KUKA KRL program: MyProgram_196().src

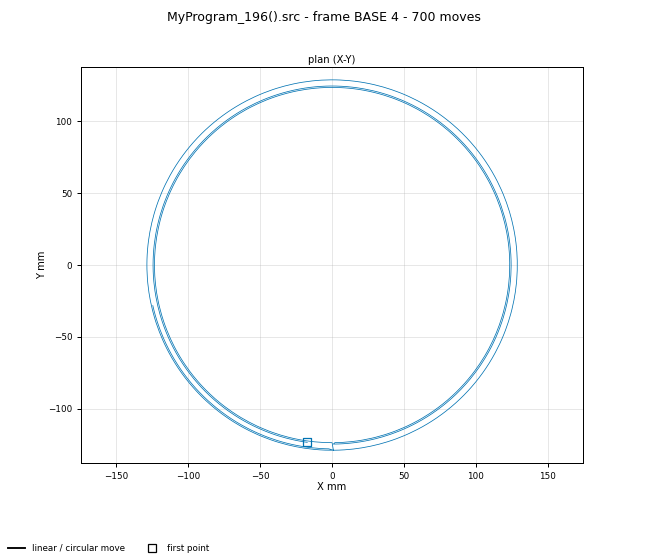
[picture p0: tool path of MyProgram_196().src in frame BASE 4, 700 of 700 moves have a stored position in this frame; points joined in program order, loops and branches not executed]
&ACCESS RVP
&REL 1
&PARAM TEMPLATE = C:\KRC\Roboter\Template\vorgabe
&PARAM EDITMASK = *
DEF MyProgram_196()
; ---- Setting reference (Base) ----
$BASE = BASE_DATA[4]

; --------------------------
; ---- Setting tool (TCP) ----
$TOOL = TOOL_DATA[3]
; --------------------------

$VEL.CP = VEL_APROX_PRINT
Startdeposition()
$VEL.CP = VEL_PRINT
LIN {X -17.3066,Y -123.2916,Z 141,A -101.2805,B 23.689,C -1.1574,E1 23.6926,E2 548.0217} C_DIS
LIN {X -20.7181,Y -122.7642,Z 141,A -102.9129,B 23.689,C -1.1559,E1 23.6881,E2 549.6594} C_DIS
LIN {X -25.1482,Y -121.934,Z 141,A -104.9652,B 23.689,C -1.1577,E1 23.6825,E2 551.7095} C_DIS
LIN {X -31.1595,Y -120.5388,Z 141,A -107.6921,B 23.6887,C -1.1643,E1 23.6751,E2 554.424} C_DIS
LIN {X -33.6692,Y -119.8608,Z 141,A -108.9963,B 23.6889,C -1.1602,E1 23.6716,E2 555.7403} C_DIS
LIN {X -36.6545,Y -118.9819,Z 141,A -110.4119,B 23.6889,C -1.162,E1 23.6678,E2 557.1541} C_DIS
LIN {X -39.4614,Y -118.0805,Z 141,A -111.8065,B 23.6889,C -1.1614,E1 23.6641,E2 558.5529} C_DIS
LIN {X -42.5428,Y -117.006,Z 141,A -113.362,B 23.6889,C -1.1604,E1 23.66,E2 560.1144} C_DIS
LIN {X -46.169,Y -115.6234,Z 141,A -115.2404,B 23.6889,C -1.158,E1 23.6551,E2 562.0028} C_DIS
LIN {X -50.7496,Y -113.6867,Z 141,A -117.3609,B 23.6885,C -1.1679,E1 23.6497,E2 564.1039} C_DIS
LIN {X -54.336,Y -112.0192,Z 141,A -119.1495,B 23.6884,C -1.1715,E1 23.6452,E2 565.8885} C_DIS
LIN {X -57.8725,Y -110.2313,Z 141,A -120.9361,B 23.6882,C -1.1755,E1 23.6407,E2 567.6703} C_DIS
LIN {X -61.1046,Y -108.4752,Z 141,A -122.7725,B 23.6884,C -1.1715,E1 23.6362,E2 569.5223} C_DIS
LIN {X -64.9923,Y -106.1916,Z 141,A -124.5928,B 23.6877,C -1.1857,E1 23.6319,E2 571.313} C_DIS
LIN {X -67.5246,Y -104.6,Z 141,A -126.2397,B 23.6882,C -1.176,E1 23.628,E2 572.9897} C_DIS
LIN {X -71.7527,Y -101.7456,Z 141,A -128.2349,B 23.6872,C -1.1952,E1 23.6235,E2 574.9438} C_DIS
LIN {X -75.0263,Y -99.3563,Z 141,A -130.4687,B 23.6879,C -1.1824,E1 23.6183,E2 577.218} C_DIS
LIN {X -78.4831,Y -96.6498,Z 141,A -132.5143,B 23.6877,C -1.1851,E1 23.6139,E2 579.2651} C_DIS
LIN {X -81.6923,Y -93.9523,Z 141,A -134.4843,B 23.6877,C -1.1871,E1 23.6097,E2 581.2382} C_DIS
LIN {X -85.1342,Y -90.8457,Z 141,A -136.6203,B 23.6874,C -1.1913,E1 23.6053,E2 583.3728} C_DIS
LIN {X -88.2078,Y -87.8637,Z 141,A -138.5647,B 23.6872,C -1.1967,E1 23.6014,E2 585.3126} C_DIS
LIN {X -91.1663,Y -84.79,Z 141,A -140.5025,B 23.6869,C -1.2021,E1 23.5977,E2 587.2457} C_DIS
LIN {X -94.3561,Y -81.2253,Z 141,A -142.5001,B 23.6863,C -1.2158,E1 23.5941,E2 589.2185} C_DIS
LIN {X -96.0854,Y -79.1726,Z 141,A -144.0072,B 23.6867,C -1.2071,E1 23.5913,E2 590.7547} C_DIS
LIN {X -98.6893,Y -75.9024,Z 141,A -145.9776,B 23.6866,C -1.2098,E1 23.5879,E2 592.7283} C_DIS
LIN {X -101.3019,Y -72.3779,Z 141,A -148.129,B 23.6866,C -1.2092,E1 23.5844,E2 594.8922} C_DIS
LIN {X -103.9608,Y -68.5039,Z 141,A -150.1422,B 23.686,C -1.2211,E1 23.5813,E2 596.8864} C_DIS
LIN {X -106.2239,Y -64.9397,Z 141,A -152.0556,B 23.6857,C -1.2275,E1 23.5785,E2 598.7942} C_DIS
LIN {X -108.3531,Y -61.3219,Z 141,A -154.0839,B 23.6857,C -1.2286,E1 23.5756,E2 600.8308} C_DIS
LIN {X -110.493,Y -57.374,Z 141,A -155.9511,B 23.6849,C -1.2428,E1 23.5732,E2 602.6732} C_DIS
LIN {X -112.6362,Y -53.0445,Z 141,A -158.2325,B 23.6848,C -1.2465,E1 23.5704,E2 604.9581} C_DIS
LIN {X -114.2456,Y -49.4785,Z 141,A -160.0905,B 23.6846,C -1.2493,E1 23.5683,E2 606.82} C_DIS
LIN {X -115.6132,Y -46.1941,Z 141,A -161.8382,B 23.6846,C -1.2495,E1 23.5664,E2 608.5777} C_DIS
LIN {X -117.0709,Y -42.3627,Z 141,A -163.641,B 23.6842,C -1.2586,E1 23.5647,E2 610.3685} C_DIS
LIN {X -118.1962,Y -39.114,Z 141,A -165.24,B 23.684,C -1.2626,E1 23.5632,E2 611.967} C_DIS
LIN {X -119.7022,Y -34.2364,Z 141,A -167.5392,B 23.6835,C -1.2718,E1 23.5614,E2 614.2573} C_DIS
LIN {X -120.5071,Y -31.2844,Z 141,A -168.9347,B 23.6832,C -1.2767,E1 23.5604,E2 615.6491} C_DIS
LIN {X -121.2131,Y -28.4269,Z 141,A -170.8638,B 23.6842,C -1.257,E1 23.5591,E2 617.6396} C_DIS
LIN {X -122.0549,Y -24.5539,Z 141,A -171.9959,B 23.6825,C -1.2915,E1 23.5585,E2 618.6924} C_DIS
LIN {X -122.5458,Y -21.9722,Z 141,A -173.9291,B 23.6838,C -1.2653,E1 23.5575,E2 620.7035} C_DIS
LIN {X -123.2084,Y -17.8892,Z 141,A -175.3683,B 23.6825,C -1.2905,E1 23.557,E2 622.0886} C_DIS
LIN {X -123.6579,Y -14.4595,Z 141,A -176.892,B 23.6821,C -1.2984,E1 23.5564,E2 623.6022} C_DIS
LIN {X -123.9664,Y -11.5209,Z 141,A -178.4267,B 23.6823,C -1.2955,E1 23.556,E2 625.1539} C_DIS
LIN {X -124.2836,Y -7.3465,Z 141,A 179.8305,B 23.6816,C -1.3093,E1 23.5557,E2 626.8732} C_DIS
LIN {X -124.4226,Y -4.4158,Z 141,A 178.2604,B 23.6818,C -1.3046,E1 23.5555,E2 628.4653} C_DIS
LIN {X -124.5041,Y 0,Z 141,A 176.192,B 23.6815,C -1.3096,E1 23.5555,E2 630.5343} C_DIS
LIN {X -124.4406,Y 3.8734,Z 141,A 174.6213,B 23.6808,C -1.3242,E1 23.5555,E2 632.0784} C_DIS
LIN {X -124.2882,Y 7.271,Z 141,A 172.9166,B 23.6808,C -1.3235,E1 23.5558,E2 633.7958} C_DIS
LIN {X -124.0047,Y 11.1136,Z 141,A 170.7128,B 23.6815,C -1.3115,E1 23.5563,E2 636.0437} C_DIS
LIN {X -123.6032,Y 14.9174,Z 141,A 168.4748,B 23.6822,C -1.2977,E1 23.5571,E2 638.3305} C_DIS
LIN {X -122.7092,Y 21.0481,Z 141,A 166.196,B 23.6805,C -1.3303,E1 23.5581,E2 640.542} C_DIS
LIN {X -122.1083,Y 24.2919,Z 141,A 164.8985,B 23.6797,C -1.3443,E1 23.5588,E2 641.8126} C_DIS
LIN {X -121.1947,Y 28.503,Z 141,A 162.8874,B 23.6794,C -1.3495,E1 23.56,E2 643.8233} C_DIS
LIN {X -120.2681,Y 32.1841,Z 141,A 161.2198,B 23.679,C -1.3583,E1 23.5612,E2 645.4791} C_DIS
LIN {X -119.4143,Y 35.2207,Z 141,A 159.7511,B 23.6788,C -1.3622,E1 23.5623,E2 646.947} C_DIS
LIN {X -118.4127,Y 38.4576,Z 141,A 158.2228,B 23.6784,C -1.3684,E1 23.5636,E2 648.4692} C_DIS
LIN {X -117.5027,Y 41.1515,Z 141,A 156.9647,B 23.6781,C -1.3746,E1 23.5648,E2 649.7193} C_DIS
LIN {X -116.5143,Y 43.8707,Z 141,A 155.022,B 23.6792,C -1.3535,E1 23.5667,E2 651.7266} C_DIS
LIN {X -114.9502,Y 47.8189,Z 141,A 153.8518,B 23.6771,C -1.3919,E1 23.5679,E2 652.8074} C_DIS
LIN {X -113.6029,Y 50.9369,Z 141,A 151.9527,B 23.6776,C -1.3827,E1 23.57,E2 654.7407} C_DIS
LIN {X -112.2654,Y 53.8206,Z 141,A 150.502,B 23.6774,C -1.3876,E1 23.5718,E2 656.1875} C_DIS
LIN {X -110.5566,Y 57.2529,Z 141,A 148.7321,B 23.6771,C -1.3926,E1 23.574,E2 657.955} C_DIS
LIN {X -108.919,Y 60.3099,Z 141,A 146.6227,B 23.678,C -1.376,E1 23.5769,E2 660.1177} C_DIS
LIN {X -106.7792,Y 64.0229,Z 141,A 145.3003,B 23.6762,C -1.4086,E1 23.5787,E2 661.3657} C_DIS
LIN {X -105.139,Y 66.682,Z 141,A 143.6415,B 23.6765,C -1.4035,E1 23.5812,E2 663.0464} C_DIS
LIN {X -102.8195,Y 70.2058,Z 141,A 141.6627,B 23.6763,C -1.4074,E1 23.5842,E2 665.0259} C_DIS
LIN {X -100.2413,Y 73.8399,Z 141,A 139.749,B 23.6756,C -1.4187,E1 23.5873,E2 666.9211} C_DIS
LIN {X -98.1212,Y 76.6353,Z 141,A 137.9549,B 23.6758,C -1.4155,E1 23.5904,E2 668.7323} C_DIS
LIN {X -95.2628,Y 80.1602,Z 141,A 135.9027,B 23.6754,C -1.4225,E1 23.5941,E2 670.777} C_DIS
LIN {X -92.4463,Y 83.3933,Z 141,A 133.9366,B 23.6751,C -1.4278,E1 23.5977,E2 672.7392} C_DIS
LIN {X -89.5628,Y 86.4821,Z 141,A 131.9927,B 23.6748,C -1.4327,E1 23.6014,E2 674.6799} C_DIS
LIN {X -86.8396,Y 89.2167,Z 141,A 130.1509,B 23.6748,C -1.4342,E1 23.6051,E2 676.5262} C_DIS
LIN {X -83.8458,Y 92.0357,Z 141,A 128.2976,B 23.6744,C -1.4403,E1 23.6089,E2 678.3723} C_DIS
LIN {X -80.2512,Y 95.1865,Z 141,A 126.0391,B 23.6743,C -1.4428,E1 23.6136,E2 680.6339} C_DIS
LIN {X -76.8712,Y 97.936,Z 141,A 124.0446,B 23.674,C -1.4476,E1 23.618,E2 682.6243} C_DIS
LIN {X -73.4057,Y 100.5603,Z 141,A 121.9863,B 23.6739,C -1.4493,E1 23.6226,E2 684.6862} C_DIS
LIN {X -69.956,Y 102.9894,Z 141,A 120.0614,B 23.6736,C -1.4539,E1 23.627,E2 686.6065} C_DIS
LIN {X -66.1231,Y 105.4917,Z 141,A 117.6109,B 23.6742,C -1.4433,E1 23.6329,E2 689.0918} C_DIS
LIN {X -62.8782,Y 107.457,Z 141,A 115.78,B 23.6742,C -1.4428,E1 23.6373,E2 690.9298} C_DIS
LIN {X -59.2115,Y 109.5205,Z 141,A 114.2417,B 23.6731,C -1.463,E1 23.641,E2 692.4221} C_DIS
LIN {X -53.1473,Y 112.5871,Z 141,A 111.2946,B 23.6723,C -1.4758,E1 23.6483,E2 695.3456} C_DIS
LIN {X -50.7226,Y 113.6987,Z 141,A 109.9492,B 23.6725,C -1.4726,E1 23.6517,E2 696.7024} C_DIS
LIN {X -47.7132,Y 114.9944,Z 141,A 108.542,B 23.6721,C -1.4791,E1 23.6553,E2 698.0969} C_DIS
LIN {X -45.0235,Y 116.0736,Z 141,A 107.0366,B 23.6725,C -1.4735,E1 23.6593,E2 699.6198} C_DIS
LIN {X -41.6006,Y 117.3457,Z 141,A 105.0029,B 23.6732,C -1.4603,E1 23.6647,E2 701.6905} C_DIS
LIN {X -38.0606,Y 118.5395,Z 141,A 103.7953,B 23.6718,C -1.4845,E1 23.6678,E2 702.8401} C_DIS
LIN {X -34.6323,Y 119.5865,Z 141,A 102.079,B 23.6718,C -1.4834,E1 23.6724,E2 704.5622} C_DIS
LIN {X -30.8263,Y 120.6234,Z 141,A 99.7305,B 23.6731,C -1.4621,E1 23.6789,E2 706.9675} C_DIS
LIN {X -26.6986,Y 121.6043,Z 141,A 98.4667,B 23.6713,C -1.4938,E1 23.6821,E2 708.154} C_DIS
LIN {X -22.8887,Y 122.3789,Z 141,A 96.3822,B 23.672,C -1.4823,E1 23.6879,E2 710.2696} C_DIS
LIN {X -18.9799,Y 123.0448,Z 141,A 94.6737,B 23.6716,C -1.4887,E1 23.6926,E2 711.9638} C_DIS
LIN {X -15.2406,Y 123.5647,Z 141,A 92.9076,B 23.6716,C -1.4885,E1 23.6975,E2 713.7319} C_DIS
LIN {X -11.7063,Y 123.9486,Z 141,A 91.3468,B 23.6713,C -1.4927,E1 23.7018,E2 715.2833} C_DIS
LIN {X -8.1197,Y 124.2359,Z 141,A 89.5749,B 23.6716,C -1.4882,E1 23.7067,E2 717.067} C_DIS
LIN {X -4.0364,Y 124.4361,Z 141,A 87.8019,B 23.6713,C -1.4936,E1 23.7117,E2 718.827} C_DIS
LIN {X -1.1493,Y 124.4958,Z 141,A 86.3456,B 23.6716,C -1.4883,E1 23.7158,E2 720.2966} C_DIS
LIN {X 2.7069,Y 124.4724,Z 141,A 84.5293,B 23.6716,C -1.4866,E1 23.7208,E2 722.1168} C_DIS
LIN {X 6.669,Y 124.3221,Z 141,A 82.715,B 23.6716,C -1.4872,E1 23.7259,E2 723.929} C_DIS
LIN {X 10.5326,Y 124.0538,Z 141,A 81.0523,B 23.6714,C -1.4924,E1 23.7305,E2 725.5778} C_DIS
LIN {X 14.2232,Y 123.686,Z 141,A 79.2934,B 23.6715,C -1.4898,E1 23.7354,E2 727.342} C_DIS
LIN {X 17.7081,Y 123.2343,Z 141,A 77.6949,B 23.6715,C -1.4902,E1 23.7398,E2 728.9379} C_DIS
LIN {X 22.0126,Y 122.5385,Z 141,A 75.6852,B 23.6715,C -1.4894,E1 23.7453,E2 730.9475} C_DIS
LIN {X 28.4618,Y 121.2037,Z 141,A 72.786,B 23.6713,C -1.4938,E1 23.7532,E2 733.8318} C_DIS
LIN {X 31.9757,Y 120.3236,Z 141,A 71.0084,B 23.6716,C -1.4878,E1 23.7581,E2 735.6216} C_DIS
LIN {X 35.5975,Y 119.3039,Z 141,A 69.3551,B 23.6715,C -1.49,E1 23.7625,E2 737.2662} C_DIS
LIN {X 38.629,Y 118.3577,Z 141,A 67.8802,B 23.6716,C -1.4882,E1 23.7664,E2 738.7427} C_DIS
LIN {X 41.7416,Y 117.2949,Z 141,A 66.3878,B 23.6716,C -1.4879,E1 23.7703,E2 740.2328} C_DIS
LIN {X 45.712,Y 115.8059,Z 141,A 64.4266,B 23.6718,C -1.4855,E1 23.7754,E2 742.1954} C_DIS
LIN {X 48.1386,Y 114.8167,Z 141,A 63.1889,B 23.6719,C -1.4828,E1 23.7786,E2 743.4368} C_DIS
LIN {X 51.6422,Y 113.2859,Z 141,A 61.4616,B 23.6719,C -1.4822,E1 23.783,E2 745.1611} C_DIS
LIN {X 55.6591,Y 111.3671,Z 141,A 59.4544,B 23.6719,C -1.4816,E1 23.7881,E2 747.1642} C_DIS
LIN {X 59.597,Y 109.3107,Z 141,A 57.1094,B 23.673,C -1.4649,E1 23.7939,E2 749.5435} C_DIS
LIN {X 63.4067,Y 107.1465,Z 141,A 55.2096,B 23.6728,C -1.4673,E1 23.7985,E2 751.4312} C_DIS
LIN {X 66.7928,Y 105.0691,Z 141,A 53.3736,B 23.673,C -1.4641,E1 23.8029,E2 753.269} C_DIS
LIN {X 70.403,Y 102.6842,Z 141,A 51.4427,B 23.673,C -1.4636,E1 23.8073,E2 755.1942} C_DIS
LIN {X 73.2476,Y 100.6751,Z 141,A 49.9898,B 23.6728,C -1.4678,E1 23.8106,E2 756.6313} C_DIS
LIN {X 75.9908,Y 98.6212,Z 141,A 48.3246,B 23.6732,C -1.4609,E1 23.8143,E2 758.3073} C_DIS
LIN {X 79.7633,Y 95.5958,Z 141,A 46.0146,B 23.6737,C -1.4527,E1 23.8193,E2 760.6284} C_DIS
LIN {X 83.2093,Y 92.6115,Z 141,A 43.9696,B 23.6737,C -1.451,E1 23.8236,E2 762.669} C_DIS
LIN {X 86.3521,Y 89.6887,Z 141,A 41.9825,B 23.6741,C -1.4463,E1 23.8276,E2 764.6591} C_DIS
LIN {X 89.3005,Y 86.753,Z 141,A 40.1226,B 23.6741,C -1.4447,E1 23.8313,E2 766.5145} C_DIS
LIN {X 91.9746,Y 83.9131,Z 141,A 38.2695,B 23.6745,C -1.4379,E1 23.8348,E2 768.3758} C_DIS
LIN {X 94.9716,Y 80.505,Z 141,A 36.2299,B 23.6747,C -1.4354,E1 23.8385,E2 770.4119} C_DIS
LIN {X 97.6729,Y 77.2061,Z 141,A 34.236,B 23.675,C -1.4291,E1 23.842,E2 772.4113} C_DIS
LIN {X 100.3932,Y 73.6331,Z 141,A 32.3813,B 23.6747,C -1.4341,E1 23.8451,E2 774.2443} C_DIS
LIN {X 102.6283,Y 70.4845,Z 141,A 30.4624,B 23.6754,C -1.4228,E1 23.8482,E2 776.1812} C_DIS
LIN {X 104.9443,Y 66.9877,Z 141,A 28.5479,B 23.6756,C -1.4185,E1 23.8511,E2 778.0963} C_DIS
LIN {X 107.5449,Y 62.7282,Z 141,A 26.2165,B 23.6761,C -1.4107,E1 23.8545,E2 780.4343} C_DIS
LIN {X 109.7049,Y 58.8682,Z 141,A 24.1542,B 23.6765,C -1.4038,E1 23.8573,E2 782.5022} C_DIS
LIN {X 111.8497,Y 54.6808,Z 141,A 22.2107,B 23.6762,C -1.4084,E1 23.8597,E2 784.4234} C_DIS
LIN {X 113.1798,Y 51.8717,Z 141,A 20.8015,B 23.6764,C -1.4053,E1 23.8613,E2 785.8321} C_DIS
LIN {X 114.4208,Y 49.0733,Z 141,A 19.3376,B 23.6768,C -1.3986,E1 23.863,E2 787.3042} C_DIS
LIN {X 116.0662,Y 45.0425,Z 141,A 17.3425,B 23.6771,C -1.3931,E1 23.865,E2 789.3011} C_DIS
LIN {X 117.4217,Y 41.3853,Z 141,A 15.3627,B 23.6778,C -1.3788,E1 23.8669,E2 791.3045} C_DIS
LIN {X 119.9692,Y 33.2816,Z 141,A 11.7012,B 23.6778,C -1.3788,E1 23.8699,E2 794.9438} C_DIS
LIN {X 120.5954,Y 30.9366,Z 141,A 10.3603,B 23.6786,C -1.3646,E1 23.8709,E2 796.3118} C_DIS
LIN {X 121.5379,Y 27.0058,Z 141,A 8.775,B 23.6782,C -1.3721,E1 23.8718,E2 797.8689} C_DIS
LIN {X 122.4429,Y 22.5467,Z 141,A 6.549,B 23.6789,C -1.3591,E1 23.873,E2 800.1132} C_DIS
LIN {X 123.0538,Y 18.9216,Z 141,A 4.9728,B 23.6789,C -1.3593,E1 23.8737,E2 801.6789} C_DIS
LIN {X 123.6011,Y 14.9354,Z 141,A 3.0511,B 23.6794,C -1.35,E1 23.8744,E2 803.6117} C_DIS
LIN {X 124.0353,Y 10.751,Z 141,A 1.2008,B 23.6795,C -1.348,E1 23.8749,E2 805.4554} C_DIS
LIN {X 124.2915,Y 7.2182,Z 141,A -0.5168,B 23.68,C -1.3384,E1 23.8752,E2 807.1858} C_DIS
LIN {X 124.4587,Y 3.2237,Z 141,A -2.2882,B 23.6802,C -1.3358,E1 23.8754,E2 808.9525} C_DIS
LIN {X 124.5003,Y -0.6363,Z 141,A -4.0224,B 23.6804,C -1.3321,E1 23.8754,E2 810.6849} C_DIS
LIN {X 124.4376,Y -3.9818,Z 141,A -5.4713,B 23.6804,C -1.3315,E1 23.8754,E2 812.1261} C_DIS
LIN {X 124.3069,Y -6.968,Z 141,A -6.8286,B 23.6806,C -1.3279,E1 23.8751,E2 813.4838} C_DIS
LIN {X 124.109,Y -9.8786,Z 141,A -8.3348,B 23.6812,C -1.3156,E1 23.8748,E2 815.011} C_DIS
LIN {X 123.7207,Y -13.922,Z 141,A -10.1062,B 23.6813,C -1.3143,E1 23.8743,E2 816.7745} C_DIS
LIN {X 123.3029,Y -17.2276,Z 141,A -11.6455,B 23.6816,C -1.309,E1 23.8737,E2 818.3172} C_DIS
LIN {X 122.7639,Y -20.72,Z 141,A -13.2447,B 23.6818,C -1.3051,E1 23.873,E2 819.9162} C_DIS
LIN {X 121.6615,Y -26.4335,Z 141,A -16.6052,B 23.6839,C -1.2635,E1 23.8711,E2 823.3589} C_DIS
LIN {X 120.4326,Y -31.5669,Z 141,A -18.1603,B 23.6822,C -1.298,E1 23.8701,E2 824.8191} C_DIS
LIN {X 119.0643,Y -36.3852,Z 141,A -20.5726,B 23.6828,C -1.2854,E1 23.8682,E2 827.2478} C_DIS
LIN {X 118.0946,Y -39.4191,Z 141,A -22.0853,B 23.6832,C -1.2785,E1 23.8669,E2 828.7685} C_DIS
LIN {X 116.6591,Y -43.4842,Z 141,A -24.1103,B 23.6836,C -1.2703,E1 23.8649,E2 830.8017} C_DIS
LIN {X 115.3435,Y -46.8633,Z 141,A -25.5935,B 23.6834,C -1.2742,E1 23.8634,E2 832.2667} C_DIS
LIN {X 114.0457,Y -49.9409,Z 141,A -27.1788,B 23.6837,C -1.2671,E1 23.8617,E2 833.8603} C_DIS
LIN {X 111.9483,Y -54.4811,Z 141,A -29.4012,B 23.6839,C -1.2639,E1 23.8591,E2 836.0778} C_DIS
LIN {X 110.7736,Y -56.8289,Z 141,A -30.7854,B 23.6845,C -1.2518,E1 23.8573,E2 837.4842} C_DIS
LIN {X 108.6377,Y -60.8156,Z 141,A -32.8381,B 23.6847,C -1.247,E1 23.8545,E2 839.5373} C_DIS
LIN {X 106.3977,Y -64.6547,Z 141,A -34.8786,B 23.685,C -1.2413,E1 23.8516,E2 841.5808} C_DIS
LIN {X 103.7595,Y -68.8094,Z 141,A -36.9126,B 23.6848,C -1.2461,E1 23.8486,E2 843.5923} C_DIS
LIN {X 101.9788,Y -71.4219,Z 141,A -38.5838,B 23.6855,C -1.2315,E1 23.8459,E2 845.2907} C_DIS
LIN {X 99.4874,Y -74.8527,Z 141,A -40.5248,B 23.6857,C -1.2267,E1 23.8426,E2 847.2338} C_DIS
LIN {X 95.9047,Y -79.3909,Z 141,A -43.0677,B 23.6858,C -1.2253,E1 23.8382,E2 849.7676} C_DIS
LIN {X 93.457,Y -82.2586,Z 141,A -44.8721,B 23.6862,C -1.2174,E1 23.8349,E2 851.5828} C_DIS
LIN {X 89.71,Y -86.3298,Z 141,A -47.6126,B 23.6869,C -1.2017,E1 23.8296,E2 854.3495} C_DIS
LIN {X 86.2219,Y -89.8136,Z 141,A -49.6807,B 23.6867,C -1.2058,E1 23.8255,E2 856.3983} C_DIS
LIN {X 83.0138,Y -92.7865,Z 141,A -51.8253,B 23.6873,C -1.1948,E1 23.821,E2 858.561} C_DIS
LIN {X 79.4464,Y -95.8587,Z 141,A -53.6942,B 23.6868,C -1.2041,E1 23.8171,E2 860.3991} C_DIS
LIN {X 76.668,Y -98.0956,Z 141,A -55.4558,B 23.6873,C -1.1948,E1 23.8132,E2 862.1769} C_DIS
LIN {X 73.29,Y -100.6443,Z 141,A -57.3884,B 23.6874,C -1.1914,E1 23.8089,E2 864.1107} C_DIS
LIN {X 69.347,Y -103.4007,Z 141,A -59.5811,B 23.6876,C -1.1879,E1 23.8039,E2 866.3039} C_DIS
LIN {X 66.3806,Y -105.3292,Z 141,A -61.1976,B 23.6877,C -1.1853,E1 23.8,E2 867.9214} C_DIS
LIN {X 62.6977,Y -107.5628,Z 141,A -63.211,B 23.688,C -1.1802,E1 23.7952,E2 869.9409} C_DIS
LIN {X 59.2894,Y -109.4784,Z 141,A -64.9736,B 23.688,C -1.1788,E1 23.7909,E2 871.7017} C_DIS
LIN {X 56.384,Y -111,Z 141,A -66.389,B 23.688,C -1.1807,E1 23.7874,E2 873.1081} C_DIS
LIN {X 53.0972,Y -112.611,Z 141,A -68.2652,B 23.6885,C -1.1689,E1 23.7826,E2 875.0082} C_DIS
LIN {X 49.5828,Y -114.2005,Z 141,A -69.8564,B 23.6882,C -1.1749,E1 23.7786,E2 876.5805} C_DIS
LIN {X 45.9656,Y -115.7054,Z 141,A -71.7351,B 23.6885,C -1.1688,E1 23.7737,E2 878.4699} C_DIS
LIN {X 40.6054,Y -117.6921,Z 141,A -74.2803,B 23.6885,C -1.1693,E1 23.7671,E2 881.0081} C_DIS
LIN {X 35.0163,Y -119.4741,Z 141,A -77.2355,B 23.6892,C -1.1543,E1 23.7591,E2 883.9951} C_DIS
LIN {X 30.4704,Y -120.7137,Z 141,A -79.1386,B 23.6887,C -1.1643,E1 23.754,E2 885.87} C_DIS
LIN {X 27.3829,Y -121.4517,Z 141,A -80.6986,B 23.689,C -1.1583,E1 23.7497,E2 887.4425} C_DIS
LIN {X 23.3018,Y -122.2999,Z 141,A -82.5163,B 23.6888,C -1.1614,E1 23.7448,E2 889.2504} C_DIS
LIN {X 19.7091,Y -122.9319,Z 141,A -84.2865,B 23.6891,C -1.1558,E1 23.7399,E2 891.0325} C_DIS
LIN {X 15.9693,Y -123.4718,Z 141,A -85.9516,B 23.689,C -1.1581,E1 23.7353,E2 892.6903} C_DIS
LIN {X 11.9617,Y -123.9241,Z 141,A -87.7488,B 23.689,C -1.1598,E1 23.7303,E2 894.4821} C_DIS
LIN {X 8.1149,Y -124.2362,Z 141,A -89.5983,B 23.6891,C -1.1556,E1 23.7251,E2 896.3411} C_DIS
LIN {X 4.476,Y -124.4202,Z 141,A -91.1477,B 23.6889,C -1.1608,E1 23.7209,E2 897.877} C_DIS
LIN {X 0.873,Y -124.4971,Z 141,A -92.8007,B 23.6889,C -1.1606,E1 23.7162,E2 899.5302} C_DIS
Enddeposition()
LIN {X 0.873,Y -124.4971,Z 141,A -92.8007,B 23.6889,C -1.1606,E1 23.7162,E2 899.5302} C_DIS
Startdeposition()
$VEL.CP = VEL_PRINT
LIN {X 1.924,Y -123.5134,Z 141,A -91.6348,B 22.9991,C -1.0757,E1 23.0264,E2 898.4877} C_DIS
LIN {X 4.8123,Y -123.4345,Z 141,A -90.1828,B 22.9989,C -1.0811,E1 23.0305,E2 897.0222} C_DIS
LIN {X 7.5776,Y -123.2956,Z 141,A -88.8989,B 22.9989,C -1.0816,E1 23.0341,E2 895.7376} C_DIS
LIN {X 10.8747,Y -123.0495,Z 141,A -87.3807,B 22.9989,C -1.0816,E1 23.0383,E2 894.2202} C_DIS
LIN {X 13.6106,Y -122.7767,Z 141,A -86.0685,B 22.9988,C -1.084,E1 23.0419,E2 892.9028} C_DIS
LIN {X 17.4387,Y -122.291,Z 141,A -84.2404,B 22.9986,C -1.0868,E1 23.047,E2 891.0692} C_DIS
LIN {X 21.1194,Y -121.711,Z 141,A -82.57,B 22.9986,C -1.0855,E1 23.0516,E2 889.404} C_DIS
LIN {X 24.3687,Y -121.1009,Z 141,A -81.0461,B 22.9986,C -1.0863,E1 23.0558,E2 887.8799} C_DIS
LIN {X 27.0583,Y -120.529,Z 141,A -79.772,B 22.9986,C -1.0874,E1 23.0593,E2 886.6049} C_DIS
LIN {X 30.0457,Y -119.8188,Z 141,A -78.2907,B 22.9984,C -1.0914,E1 23.0633,E2 885.1158} C_DIS
LIN {X 33.175,Y -118.9898,Z 141,A -76.8671,B 22.9985,C -1.0895,E1 23.0671,E2 883.6997} C_DIS
LIN {X 35.9751,Y -118.1735,Z 141,A -75.6331,B 22.9987,C -1.0856,E1 23.0704,E2 882.478} C_DIS
LIN {X 38.2193,Y -117.4686,Z 141,A -74.2091,B 22.9979,C -1.102,E1 23.0743,E2 881.0148} C_DIS
LIN {X 41.6033,Y -116.3116,Z 141,A -72.6935,B 22.9981,C -1.0976,E1 23.0782,E2 879.5139} C_DIS
LIN {X 44.4569,Y -115.2511,Z 141,A -71.2892,B 22.9981,C -1.0992,E1 23.0819,E2 878.1089} C_DIS
LIN {X 47.5233,Y -114.0204,Z 141,A -69.8316,B 22.9981,C -1.0979,E1 23.0856,E2 876.6583} C_DIS
LIN {X 50.0486,Y -112.9355,Z 141,A -68.5647,B 22.9981,C -1.0995,E1 23.0889,E2 875.3908} C_DIS
LIN {X 53.0594,Y -111.552,Z 141,A -67.0128,B 22.9979,C -1.1025,E1 23.0928,E2 873.8354} C_DIS
LIN {X 56.2559,Y -109.9747,Z 141,A -65.3262,B 22.9977,C -1.1068,E1 23.097,E2 872.143} C_DIS
LIN {X 59.57,Y -108.2177,Z 141,A -63.5816,B 22.9976,C -1.11,E1 23.1013,E2 870.3957} C_DIS
LIN {X 62.4465,Y -106.5835,Z 141,A -62.191,B 22.9978,C -1.1061,E1 23.1047,E2 869.0197} C_DIS
LIN {X 65.1936,Y -104.9256,Z 141,A -60.6931,B 22.9976,C -1.1093,E1 23.1082,E2 867.5188} C_DIS
LIN {X 67.5932,Y -103.3967,Z 141,A -59.3186,B 22.9974,C -1.1144,E1 23.1115,E2 866.1362} C_DIS
LIN {X 70.6713,Y -101.3171,Z 141,A -57.4929,B 22.997,C -1.1226,E1 23.1157,E2 864.2964} C_DIS
LIN {X 73.8096,Y -99.0541,Z 141,A -55.7375,B 22.997,C -1.1245,E1 23.1197,E2 862.5429} C_DIS
LIN {X 77.1802,Y -96.4515,Z 141,A -53.8346,B 22.9969,C -1.1254,E1 23.1238,E2 860.6455} C_DIS
LIN {X 80.1999,Y -93.9554,Z 141,A -51.9098,B 22.9965,C -1.1345,E1 23.128,E2 858.7057} C_DIS
LIN {X 83.5157,Y -91.0204,Z 141,A -49.9777,B 22.9965,C -1.1335,E1 23.132,E2 856.7845} C_DIS
LIN {X 86.2585,Y -88.426,Z 141,A -48.1098,B 22.996,C -1.1432,E1 23.1358,E2 854.9006} C_DIS
LIN {X 89.4406,Y -85.2055,Z 141,A -46.0365,B 22.9959,C -1.1471,E1 23.1398,E2 852.8271} C_DIS
LIN {X 92.1283,Y -82.292,Z 141,A -44.2204,B 22.9957,C -1.1507,E1 23.1432,E2 851.0106} C_DIS
LIN {X 94.996,Y -78.9645,Z 141,A -42.2006,B 22.9955,C -1.1552,E1 23.1468,E2 848.9896} C_DIS
LIN {X 97.3627,Y -76.0276,Z 141,A -40.528,B 22.9955,C -1.1562,E1 23.1497,E2 847.323} C_DIS
LIN {X 99.2205,Y -73.5861,Z 141,A -39.1666,B 22.9954,C -1.1571,E1 23.152,E2 845.9662} C_DIS
LIN {X 101.1523,Y -70.9078,Z 141,A -37.6842,B 22.9953,C -1.159,E1 23.1544,E2 844.4869} C_DIS
LIN {X 102.7044,Y -68.6395,Z 141,A -36.384,B 22.9951,C -1.1638,E1 23.1564,E2 843.1817} C_DIS
LIN {X 104.7101,Y -65.5399,Z 141,A -34.7368,B 22.995,C -1.1656,E1 23.1589,E2 841.5391} C_DIS
LIN {X 105.9552,Y -63.5072,Z 141,A -33.5869,B 22.9947,C -1.1708,E1 23.1606,E2 840.3823} C_DIS
LIN {X 107.616,Y -60.6497,Z 141,A -32.0617,B 22.9945,C -1.1749,E1 23.1627,E2 838.8554} C_DIS
LIN {X 109.0694,Y -57.9946,Z 141,A -30.6738,B 22.9944,C -1.1783,E1 23.1645,E2 837.4669} C_DIS
LIN {X 110.5616,Y -55.0952,Z 141,A -29.2696,B 22.9944,C -1.1776,E1 23.1663,E2 836.0724} C_DIS
LIN {X 111.7978,Y -52.5448,Z 141,A -27.8512,B 22.994,C -1.1865,E1 23.168,E2 834.6399} C_DIS
LIN {X 112.9347,Y -50.0505,Z 141,A -26.591,B 22.9938,C -1.1898,E1 23.1695,E2 833.3787} C_DIS
LIN {X 114.1794,Y -47.1426,Z 141,A -25.1245,B 22.9936,C -1.1943,E1 23.1711,E2 831.9098} C_DIS
LIN {X 115.6044,Y -43.5292,Z 141,A -23.5727,B 22.9939,C -1.188,E1 23.1726,E2 830.3833} C_DIS
LIN {X 116.3059,Y -41.6192,Z 141,A -22.3342,B 22.9931,C -1.2049,E1 23.1738,E2 829.1095} C_DIS
LIN {X 117.3819,Y -38.4831,Z 141,A -20.9021,B 22.9931,C -1.2046,E1 23.1751,E2 827.6868} C_DIS
LIN {X 118.2075,Y -35.864,Z 141,A -19.6181,B 22.9929,C -1.2091,E1 23.1761,E2 826.3994} C_DIS
LIN {X 119.0554,Y -32.9406,Z 141,A -18.1951,B 22.9926,C -1.2141,E1 23.1772,E2 824.9727} C_DIS
LIN {X 119.8908,Y -29.7621,Z 141,A -16.7106,B 22.9925,C -1.2171,E1 23.1782,E2 823.4901} C_DIS
LIN {X 120.5202,Y -27.0966,Z 141,A -15.4496,B 22.9923,C -1.2207,E1 23.179,E2 822.228} C_DIS
LIN {X 121.1923,Y -23.9194,Z 141,A -13.9064,B 22.9919,C -1.2272,E1 23.1799,E2 820.678} C_DIS
LIN {X 121.81,Y -20.5321,Z 141,A -12.3343,B 22.9917,C -1.2312,E1 23.1807,E2 819.1059} C_DIS
LIN {X 122.4067,Y -16.6169,Z 141,A -10.449,B 22.9913,C -1.2394,E1 23.1814,E2 817.2119} C_DIS
LIN {X 122.7765,Y -13.6122,Z 141,A -9.1362,B 22.9913,C -1.2396,E1 23.1818,E2 815.9071} C_DIS
LIN {X 123.0963,Y -10.3208,Z 141,A -7.6271,B 22.9911,C -1.2434,E1 23.1822,E2 814.3981} C_DIS
LIN {X 123.2956,Y -7.5781,Z 141,A -6.3596,B 22.9909,C -1.2471,E1 23.1824,E2 813.1294} C_DIS
LIN {X 123.4561,Y -4.258,Z 141,A -4.8605,B 22.9908,C -1.2501,E1 23.1826,E2 811.6326} C_DIS
LIN {X 123.5248,Y -1.1038,Z 141,A -3.5741,B 22.991,C -1.2464,E1 23.1826,E2 810.364} C_DIS
LIN {X 123.5156,Y 1.7938,Z 141,A -1.9532,B 22.9901,C -1.2639,E1 23.1826,E2 808.7092} C_DIS
LIN {X 123.4342,Y 4.8198,Z 141,A -0.5126,B 22.9897,C -1.2701,E1 23.1826,E2 807.2621} C_DIS
LIN {X 123.1932,Y 9.0924,Z 141,A 1.3573,B 22.9897,C -1.271,E1 23.1822,E2 805.4021} C_DIS
LIN {X 122.9069,Y 12.3875,Z 141,A 2.8213,B 22.9897,C -1.2726,E1 23.1818,E2 803.9436} C_DIS
LIN {X 122.5669,Y 15.395,Z 141,A 4.378,B 22.989,C -1.2843,E1 23.1813,E2 802.3672} C_DIS
LIN {X 122.0573,Y 19.0061,Z 141,A 5.9649,B 22.989,C -1.2847,E1 23.1806,E2 800.7895} C_DIS
LIN {X 121.4422,Y 22.6126,Z 141,A 7.6964,B 22.9886,C -1.2916,E1 23.1798,E2 799.0515} C_DIS
LIN {X 120.7918,Y 25.8566,Z 141,A 9.0456,B 22.9888,C -1.2877,E1 23.179,E2 797.721} C_DIS
LIN {X 120.1785,Y 28.5736,Z 141,A 10.4106,B 22.9884,C -1.2951,E1 23.1781,E2 796.3457} C_DIS
LIN {X 119.3795,Y 31.7443,Z 141,A 11.9149,B 22.9882,C -1.2992,E1 23.1771,E2 794.8406} C_DIS
LIN {X 118.577,Y 34.6214,Z 141,A 13.2879,B 22.988,C -1.3028,E1 23.176,E2 793.467} C_DIS
LIN {X 117.7932,Y 37.2031,Z 141,A 14.5852,B 22.9877,C -1.3087,E1 23.1749,E2 792.1626} C_DIS
LIN {X 116.7167,Y 40.4519,Z 141,A 16.0415,B 22.9877,C -1.3073,E1 23.1737,E2 790.719} C_DIS
LIN {X 115.6907,Y 43.2988,Z 141,A 17.5528,B 22.9873,C -1.3165,E1 23.1722,E2 789.1935} C_DIS
LIN {X 114.5954,Y 46.1195,Z 141,A 19.0266,B 22.9869,C -1.324,E1 23.1707,E2 787.7097} C_DIS
LIN {X 112.9302,Y 50.0606,Z 141,A 20.8698,B 22.9869,C -1.323,E1 23.1686,E2 785.88} C_DIS
LIN {X 111.5493,Y 53.065,Z 141,A 22.4002,B 22.9867,C -1.3272,E1 23.1668,E2 784.3479} C_DIS
LIN {X 110.3342,Y 55.5497,Z 141,A 23.6639,B 22.9865,C -1.3299,E1 23.1652,E2 783.0848} C_DIS
LIN {X 108.8495,Y 58.4068,Z 141,A 25.0997,B 22.9865,C -1.3313,E1 23.1634,E2 781.6537} C_DIS
LIN {X 107.2707,Y 61.2583,Z 141,A 26.6218,B 22.9862,C -1.3359,E1 23.1613,E2 780.1286} C_DIS
LIN {X 105.9638,Y 63.4927,Z 141,A 28.0025,B 22.9856,C -1.3475,E1 23.1593,E2 778.7262} C_DIS
LIN {X 104.0834,Y 66.5299,Z 141,A 29.4239,B 22.9859,C -1.3409,E1 23.1572,E2 777.3294} C_DIS
LIN {X 102.5566,Y 68.8609,Z 141,A 30.9137,B 22.9852,C -1.3534,E1 23.1549,E2 775.8158} C_DIS
LIN {X 100.1127,Y 72.3674,Z 141,A 32.8638,B 22.9851,C -1.3569,E1 23.1517,E2 773.8674} C_DIS
LIN {X 97.7651,Y 75.5089,Z 141,A 34.685,B 22.9848,C -1.3615,E1 23.1486,E2 772.044} C_DIS
LIN {X 95.4084,Y 78.4663,Z 141,A 36.4732,B 22.9845,C -1.3672,E1 23.1455,E2 770.2502} C_DIS
LIN {X 92.5374,Y 81.8316,Z 141,A 38.4724,B 22.9843,C -1.3695,E1 23.1418,E2 768.255} C_DIS
LIN {X 89.888,Y 84.7332,Z 141,A 40.2805,B 22.9842,C -1.373,E1 23.1384,E2 766.4469} C_DIS
LIN {X 86.8115,Y 87.8833,Z 141,A 42.3581,B 22.9838,C -1.379,E1 23.1343,E2 764.3638} C_DIS
LIN {X 83.625,Y 90.9199,Z 141,A 44.281,B 22.9838,C -1.3777,E1 23.1304,E2 762.4526} C_DIS
LIN {X 80.7949,Y 93.4442,Z 141,A 46.1286,B 22.9835,C -1.3853,E1 23.1265,E2 760.5938} C_DIS
LIN {X 77.2902,Y 96.3634,Z 141,A 48.107,B 22.9835,C -1.383,E1 23.1223,E2 758.6294} C_DIS
LIN {X 74.7965,Y 98.3115,Z 141,A 49.6792,B 22.9832,C -1.3905,E1 23.1187,E2 757.0445} C_DIS
LIN {X 71.3624,Y 100.8316,Z 141,A 51.7132,B 22.9828,C -1.3966,E1 23.1141,E2 755.0028} C_DIS
LIN {X 67.5977,Y 103.3938,Z 141,A 53.748,B 22.9828,C -1.3965,E1 23.1094,E2 752.9756} C_DIS
LIN {X 64.5669,Y 105.3123,Z 141,A 55.2022,B 22.9832,C -1.3896,E1 23.106,E2 751.5442} C_DIS
LIN {X 62.2078,Y 106.7235,Z 141,A 56.622,B 22.9827,C -1.398,E1 23.1026,E2 750.1077} C_DIS
LIN {X 59.3142,Y 108.3579,Z 141,A 58.0973,B 22.9827,C -1.3972,E1 23.099,E2 748.6392} C_DIS
LIN {X 56.6472,Y 109.7755,Z 141,A 59.4469,B 22.9827,C -1.3967,E1 23.0956,E2 747.2949} C_DIS
LIN {X 54.1925,Y 111.0069,Z 141,A 60.8358,B 22.9824,C -1.4035,E1 23.0921,E2 745.8926} C_DIS
LIN {X 51.1882,Y 112.4251,Z 141,A 62.2874,B 22.9825,C -1.4013,E1 23.0885,E2 744.4507} C_DIS
LIN {X 48.2638,Y 113.7112,Z 141,A 63.9743,B 22.9819,C -1.4122,E1 23.0841,E2 742.7405} C_DIS
LIN {X 44.4513,Y 115.2533,Z 141,A 65.6965,B 22.9823,C -1.4058,E1 23.0797,E2 741.0387} C_DIS
LIN {X 41.6142,Y 116.3077,Z 141,A 67.0678,B 22.9823,C -1.4058,E1 23.0761,E2 739.6709} C_DIS
LIN {X 38.4895,Y 117.3798,Z 141,A 68.5786,B 22.9823,C -1.406,E1 23.0721,E2 738.1625} C_DIS
LIN {X 35.867,Y 118.2066,Z 141,A 69.8688,B 22.9822,C -1.4077,E1 23.0686,E2 736.8706} C_DIS
LIN {X 32.9612,Y 119.0496,Z 141,A 71.2959,B 22.982,C -1.4098,E1 23.0648,E2 735.4409} C_DIS
LIN {X 29.2546,Y 120.0143,Z 141,A 72.9917,B 22.9822,C -1.4073,E1 23.0602,E2 733.7542} C_DIS
LIN {X 25.9165,Y 120.7789,Z 141,A 74.722,B 22.9818,C -1.4144,E1 23.0555,E2 732.0082} C_DIS
LIN {X 22.3385,Y 121.4929,Z 141,A 76.3315,B 22.9819,C -1.4114,E1 23.0511,E2 730.4083} C_DIS
LIN {X 18.9776,Y 122.0616,Z 141,A 77.934,B 22.9819,C -1.4129,E1 23.0467,E2 728.8037} C_DIS
LIN {X 15.3233,Y 122.576,Z 141,A 79.6953,B 22.9817,C -1.4155,E1 23.0418,E2 727.0375} C_DIS
LIN {X 12.1082,Y 122.9337,Z 141,A 81.1813,B 22.9817,C -1.4151,E1 23.0377,E2 725.5535} C_DIS
LIN {X 8.8142,Y 123.2135,Z 141,A 82.7531,B 22.9817,C -1.4169,E1 23.0333,E2 723.978} C_DIS
LIN {X 4.8268,Y 123.4339,Z 141,A 84.5392,B 22.9817,C -1.414,E1 23.0283,E2 722.2} C_DIS
LIN {X 1.2335,Y 123.5234,Z 141,A 86.0805,B 22.9821,C -1.4083,E1 23.024,E2 720.6736} C_DIS
LIN {X -1.7932,Y 123.5156,Z 141,A 87.4975,B 22.9821,C -1.4086,E1 23.0201,E2 719.2557} C_DIS
LIN {X -4.8194,Y 123.4342,Z 141,A 88.9743,B 22.9819,C -1.4114,E1 23.0159,E2 717.7716} C_DIS
LIN {X -8.4149,Y 123.2426,Z 141,A 90.7815,B 22.9816,C -1.4167,E1 23.0109,E2 715.9503} C_DIS
LIN {X -12.386,Y 122.907,Z 141,A 92.4713,B 22.9821,C -1.409,E1 23.0062,E2 714.2793} C_DIS
LIN {X -15.3957,Y 122.5668,Z 141,A 93.8651,B 22.9821,C -1.4077,E1 23.0024,E2 712.8877} C_DIS
LIN {X -18.1176,Y 122.194,Z 141,A 95.1686,B 22.9821,C -1.4082,E1 22.9988,E2 711.5819} C_DIS
LIN {X -21.6653,Y 121.6133,Z 141,A 96.7844,B 22.9823,C -1.4048,E1 22.9943,E2 709.973} C_DIS
LIN {X -24.3738,Y 121.0998,Z 141,A 98.1351,B 22.9823,C -1.4068,E1 22.9906,E2 708.6154} C_DIS
LIN {X -27.8872,Y 120.3396,Z 141,A 99.9486,B 22.9819,C -1.4116,E1 22.9856,E2 706.7871} C_DIS
LIN {X -31.7604,Y 119.3752,Z 141,A 101.7733,B 22.9821,C -1.4087,E1 22.9807,E2 704.9671} C_DIS
LIN {X -36.118,Y 118.1297,Z 141,A 103.8012,B 22.9824,C -1.4033,E1 22.9753,E2 702.9494} C_DIS
LIN {X -38.9958,Y 117.2112,Z 141,A 105.1703,B 22.9826,C -1.4003,E1 22.9717,E2 701.5852} C_DIS
LIN {X -42.5434,Y 115.9727,Z 141,A 107.0688,B 22.9823,C -1.4046,E1 22.9666,E2 699.6713} C_DIS
LIN {X -45.8689,Y 114.6965,Z 141,A 108.6473,B 22.9826,C -1.3993,E1 22.9626,E2 698.1027} C_DIS
LIN {X -48.9221,Y 113.4273,Z 141,A 110.1004,B 22.983,C -1.3938,E1 22.9589,E2 696.6602} C_DIS
LIN {X -51.4354,Y 112.3108,Z 141,A 111.4718,B 22.9828,C -1.3959,E1 22.9553,E2 695.2796} C_DIS
LIN {X -54.4476,Y 110.8811,Z 141,A 112.8442,B 22.9834,C -1.3862,E1 22.9519,E2 693.9283} C_DIS
LIN {X -57.0167,Y 109.5829,Z 141,A 114.2049,B 22.9834,C -1.3851,E1 22.9486,E2 692.5664} C_DIS
LIN {X -59.5495,Y 108.2291,Z 141,A 115.6911,B 22.9832,C -1.3893,E1 22.9449,E2 691.0649} C_DIS
LIN {X -62.402,Y 106.6096,Z 141,A 117.0888,B 22.9837,C -1.3814,E1 22.9415,E2 689.6828} C_DIS
LIN {X -64.7523,Y 105.1986,Z 141,A 118.5695,B 22.9833,C -1.3878,E1 22.938,E2 688.1806} C_DIS
LIN {X -68.3521,Y 102.8962,Z 141,A 120.5305,B 22.9836,C -1.3832,E1 22.9334,E2 686.2246} C_DIS
LIN {X -71.3635,Y 100.8309,Z 141,A 122.1249,B 22.984,C -1.3757,E1 22.9298,E2 684.6434} C_DIS
LIN {X -73.8122,Y 99.0522,Z 141,A 123.6571,B 22.9839,C -1.3781,E1 22.9263,E2 683.099} C_DIS
LIN {X -77.1859,Y 96.447,Z 141,A 125.5426,B 22.9843,C -1.3701,E1 22.9222,E2 681.2265} C_DIS
LIN {X -80.2102,Y 93.9466,Z 141,A 127.4878,B 22.9843,C -1.3713,E1 22.918,E2 679.27} C_DIS
LIN {X -83.4159,Y 91.1121,Z 141,A 129.4085,B 22.9846,C -1.3641,E1 22.914,E2 677.3594} C_DIS
LIN {X -86.267,Y 88.4176,Z 141,A 131.3297,B 22.9846,C -1.364,E1 22.9101,E2 675.4298} C_DIS
LIN {X -89.4577,Y 85.1877,Z 141,A 133.4288,B 22.985,C -1.3586,E1 22.9061,E2 673.3346} C_DIS
LIN {X -92.1304,Y 82.2897,Z 141,A 135.2612,B 22.9852,C -1.3542,E1 22.9026,E2 671.5046} C_DIS
LIN {X -95.0035,Y 78.9553,Z 141,A 137.3091,B 22.9855,C -1.3492,E1 22.8989,E2 669.4594} C_DIS
LIN {X -97.6584,Y 75.6466,Z 141,A 139.0515,B 22.9863,C -1.3348,E1 22.896,E2 667.7449} C_DIS
LIN {X -99.2219,Y 73.5842,Z 141,A 140.3753,B 22.9862,C -1.3366,E1 22.8937,E2 666.4095} C_DIS
LIN {X -101.1542,Y 70.9051,Z 141,A 141.8774,B 22.9865,C -1.3312,E1 22.8913,E2 664.9132} C_DIS
LIN {X -102.707,Y 68.6356,Z 141,A 143.1947,B 22.9865,C -1.3294,E1 22.8893,E2 663.5934} C_DIS
LIN {X -104.7231,Y 65.5189,Z 141,A 144.8645,B 22.987,C -1.3224,E1 22.8868,E2 661.9323} C_DIS
LIN {X -105.972,Y 63.479,Z 141,A 146.0401,B 22.987,C -1.322,E1 22.885,E2 660.7513} C_DIS
LIN {X -107.6301,Y 60.6247,Z 141,A 147.5846,B 22.9872,C -1.3181,E1 22.8829,E2 659.2079} C_DIS
LIN {X -109.0796,Y 57.9752,Z 141,A 148.9881,B 22.9874,C -1.3141,E1 22.881,E2 657.8064} C_DIS
LIN {X -110.34,Y 55.5383,Z 141,A 150.2853,B 22.9876,C -1.3114,E1 22.8794,E2 656.5086} C_DIS
LIN {X -111.7852,Y 52.5713,Z 141,A 151.8278,B 22.9878,C -1.3073,E1 22.8775,E2 654.9675} C_DIS
LIN {X -112.9405,Y 50.0375,Z 141,A 153.1221,B 22.988,C -1.3035,E1 22.8761,E2 653.6751} C_DIS
LIN {X -114.1146,Y 47.2978,Z 141,A 154.539,B 22.9881,C -1.3007,E1 22.8745,E2 652.2568} C_DIS
LIN {X -115.2161,Y 44.5468,Z 141,A 156.0485,B 22.9881,C -1.302,E1 22.873,E2 650.7347} C_DIS
LIN {X -116.7188,Y 40.4457,Z 141,A 158.0233,B 22.9885,C -1.2937,E1 22.8711,E2 648.7691} C_DIS
LIN {X -117.7627,Y 37.2987,Z 141,A 159.4863,B 22.9889,C -1.2858,E1 22.8699,E2 647.3171} C_DIS
LIN {X -118.6414,Y 34.4017,Z 141,A 160.8998,B 22.9891,C -1.2818,E1 22.8688,E2 645.905} C_DIS
LIN {X -119.5205,Y 31.2154,Z 141,A 162.441,B 22.9894,C -1.2773,E1 22.8677,E2 644.3656} C_DIS
LIN {X -120.2494,Y 28.2794,Z 141,A 163.8473,B 22.9896,C -1.273,E1 22.8667,E2 642.9615} C_DIS
LIN {X -120.8483,Y 25.595,Z 141,A 165.1773,B 22.9896,C -1.2711,E1 22.866,E2 641.6276} C_DIS
LIN {X -121.5113,Y 22.2354,Z 141,A 166.7168,B 22.9901,C -1.2641,E1 22.8652,E2 640.0963} C_DIS
LIN {X -122.0022,Y 19.3618,Z 141,A 168.1116,B 22.9901,C -1.2614,E1 22.8645,E2 638.6991} C_DIS
LIN {X -122.4163,Y 16.5439,Z 141,A 169.489,B 22.9903,C -1.2595,E1 22.864,E2 637.3177} C_DIS
LIN {X -122.7689,Y 13.6834,Z 141,A 170.7923,B 22.9906,C -1.2538,E1 22.8636,E2 636.0204} C_DIS
LIN {X -123.0958,Y 10.3268,Z 141,A 172.4151,B 22.9907,C -1.2512,E1 22.8632,E2 634.3938} C_DIS
LIN {X -123.3799,Y 6.0551,Z 141,A 174.3863,B 22.9911,C -1.2442,E1 22.8628,E2 632.4275} C_DIS
LIN {X -123.5112,Y 2.0561,Z 141,A 176.2458,B 22.9914,C -1.2383,E1 22.8627,E2 630.5708} C_DIS
LIN {X -123.5156,Y -1.7922,Z 141,A 177.9556,B 22.9918,C -1.2296,E1 22.8627,E2 628.8723} C_DIS
LIN {X -123.431,Y -4.9034,Z 141,A 179.4682,B 22.9919,C -1.2277,E1 22.8629,E2 627.3544} C_DIS
LIN {X -123.2956,Y -7.5775,Z 141,A -179.2654,B 22.9921,C -1.2247,E1 22.8631,E2 626.0874} C_DIS
LIN {X -123.0495,Y -10.8749,Z 141,A -177.7341,B 22.9923,C -1.2197,E1 22.8634,E2 624.5588} C_DIS
LIN {X -122.7766,Y -13.6111,Z 141,A -176.41,B 22.9924,C -1.2177,E1 22.8638,E2 623.2314} C_DIS
LIN {X -122.3441,Y -17.067,Z 141,A -174.9528,B 22.993,C -1.2062,E1 22.8643,E2 621.7943} C_DIS
LIN {X -121.9581,Y -19.6443,Z 141,A -173.5811,B 22.9929,C -1.2089,E1 22.8649,E2 620.4064} C_DIS
LIN {X -121.334,Y -23.1784,Z 141,A -171.9889,B 22.9933,C -1.2008,E1 22.8657,E2 618.8248} C_DIS
LIN {X -120.7946,Y -25.8433,Z 141,A -170.573,B 22.9932,C -1.2032,E1 22.8665,E2 617.3937} C_DIS
LIN {X -120.1856,Y -28.5442,Z 141,A -169.3462,B 22.9935,C -1.1968,E1 22.8673,E2 616.1752} C_DIS
LIN {X -119.3786,Y -31.7477,Z 141,A -167.806,B 22.9937,C -1.1925,E1 22.8684,E2 614.6364} C_DIS
LIN {X -118.5654,Y -34.6611,Z 141,A -166.2871,B 22.9937,C -1.1929,E1 22.8695,E2 613.1067} C_DIS
LIN {X -117.2043,Y -39.0164,Z 141,A -164.2623,B 22.9941,C -1.1829,E1 22.8713,E2 611.0951} C_DIS
LIN {X -116.3078,Y -41.6138,Z 141,A -162.9097,B 22.9941,C -1.1822,E1 22.8725,E2 609.7357} C_DIS
LIN {X -114.8436,Y -45.5038,Z 141,A -160.9094,B 22.9943,C -1.1795,E1 22.8745,E2 607.73} C_DIS
LIN {X -113.4188,Y -48.9419,Z 141,A -159.3862,B 22.9949,C -1.1663,E1 22.8762,E2 606.2317} C_DIS
LIN {X -112.3072,Y -51.4431,Z 141,A -157.947,B 22.9948,C -1.1696,E1 22.8779,E2 604.7753} C_DIS
LIN {X -110.896,Y -54.4174,Z 141,A -156.4823,B 22.9951,C -1.1628,E1 22.8796,E2 603.3194} C_DIS
LIN {X -109.6493,Y -56.8902,Z 141,A -155.2172,B 22.9953,C -1.1584,E1 22.8812,E2 602.0582} C_DIS
LIN {X -108.2233,Y -59.5599,Z 141,A -153.6277,B 22.9951,C -1.1622,E1 22.8834,E2 600.4497} C_DIS
LIN {X -106.0643,Y -63.3242,Z 141,A -151.7153,B 22.9956,C -1.1527,E1 22.8861,E2 598.5509} C_DIS
LIN {X -104.1606,Y -66.4092,Z 141,A -150.0976,B 22.9959,C -1.1456,E1 22.8884,E2 596.9423} C_DIS
LIN {X -102.5587,Y -68.8578,Z 141,A -148.7385,B 22.9961,C -1.1422,E1 22.8905,E2 595.5845} C_DIS
LIN {X -100.6844,Y -71.5705,Z 141,A -147.1958,B 22.9962,C -1.1389,E1 22.893,E2 594.0419} C_DIS
LIN {X -99.0546,Y -73.8089,Z 141,A -145.7423,B 22.9961,C -1.1428,E1 22.8954,E2 592.5709} C_DIS
LIN {X -96.4496,Y -77.1826,Z 141,A -143.8262,B 22.9964,C -1.1355,E1 22.8987,E2 590.6635} C_DIS
LIN {X -93.6431,Y -80.5639,Z 141,A -141.6676,B 22.9964,C -1.1358,E1 22.9026,E2 588.4933} C_DIS
LIN {X -90.9227,Y -83.622,Z 141,A -139.7979,B 22.9966,C -1.1303,E1 22.9061,E2 586.6287} C_DIS
LIN {X -87.8845,Y -86.8102,Z 141,A -137.7074,B 22.9968,C -1.1279,E1 22.9102,E2 584.5345} C_DIS
LIN {X -84.6342,Y -89.9814,Z 141,A -135.5911,B 22.9969,C -1.1239,E1 22.9145,E2 582.4188} C_DIS
LIN {X -81.355,Y -92.9568,Z 141,A -133.627,B 22.9973,C -1.1161,E1 22.9185,E2 580.4663} C_DIS
LIN {X -78.3628,Y -95.493,Z 141,A -131.7103,B 22.9973,C -1.1167,E1 22.9227,E2 578.5398} C_DIS
LIN {X -74.8005,Y -98.3084,Z 141,A -129.7408,B 22.9977,C -1.1072,E1 22.927,E2 576.5871} C_DIS
LIN {X -71.9279,Y -100.4289,Z 141,A -128.1604,B 22.998,C -1.1011,E1 22.9305,E2 575.0161} C_DIS
LIN {X -69.912,Y -101.8425,Z 141,A -126.8298,B 22.9977,C -1.1072,E1 22.9336,E2 573.6649} C_DIS
LIN {X -66.3279,Y -104.2127,Z 141,A -124.8099,B 22.9978,C -1.1052,E1 22.9384,E2 571.6429} C_DIS
LIN {X -63.3308,Y -106.0603,Z 141,A -123.3589,B 22.9983,C -1.095,E1 22.9418,E2 570.2131} C_DIS
LIN {X -60.6446,Y -107.6189,Z 141,A -121.8565,B 22.9983,C -1.0956,E1 22.9454,E2 568.7044} C_DIS
LIN {X -57.993,Y -109.0702,Z 141,A -120.4215,B 22.9983,C -1.0952,E1 22.949,E2 567.2661} C_DIS
LIN {X -55.2711,Y -110.4749,Z 141,A -119.0486,B 22.9984,C -1.0913,E1 22.9524,E2 565.899} C_DIS
LIN {X -52.5662,Y -111.7877,Z 141,A -117.6164,B 22.9984,C -1.0913,E1 22.956,E2 564.463} C_DIS
LIN {X -50.0606,Y -112.9301,Z 141,A -116.3403,B 22.9984,C -1.0898,E1 22.9592,E2 563.1872} C_DIS
LIN {X -46.5663,Y -114.4153,Z 141,A -114.7211,B 22.9989,C -1.0818,E1 22.9634,E2 561.5844} C_DIS
LIN {X -44.4561,Y -115.2514,Z 141,A -113.4929,B 22.9986,C -1.0884,E1 22.9666,E2 560.3365} C_DIS
LIN {X -41.6189,Y -116.306,Z 141,A -112.1158,B 22.9986,C -1.086,E1 22.9702,E2 558.9626} C_DIS
LIN {X -38.4963,Y -117.3775,Z 141,A -110.6007,B 22.9988,C -1.084,E1 22.9742,E2 557.4494} C_DIS
LIN {X -35.8723,Y -118.2049,Z 141,A -109.3045,B 22.9988,C -1.084,E1 22.9777,E2 556.1509} C_DIS
LIN {X -32.4374,Y -119.1947,Z 141,A -107.6957,B 22.9989,C -1.0807,E1 22.982,E2 554.5477} C_DIS
LIN {X -29.8394,Y -119.8711,Z 141,A -106.4048,B 22.9989,C -1.0819,E1 22.9855,E2 553.2515} C_DIS
LIN {X -26.2935,Y -120.6975,Z 141,A -104.5764,B 22.9986,C -1.0872,E1 22.9905,E2 551.407} C_DIS
LIN {X -22.0009,Y -121.5533,Z 141,A -102.5994,B 22.9988,C -1.0841,E1 22.9959,E2 549.4357} C_DIS
LIN {X -18.1225,Y -122.1933,Z 141,A -100.8351,B 22.9988,C -1.0809,E1 23.0008,E2 547.6777} C_DIS
LIN {X -14.8444,Y -122.6332,Z 141,A -99.3919,B 22.9991,C -1.0767,E1 23.0048,E2 546.2443} C_DIS
LIN {X -12.1113,Y -122.9334,Z 141,A -97.9698,B 22.9988,C -1.083,E1 23.0088,E2 544.8051} C_DIS
LIN {X -8.8088,Y -123.2139,Z 141,A -96.5533,B 22.999,C -1.0776,E1 23.0127,E2 543.4018} C_DIS
LIN {X -6.0646,Y -123.3794,Z 141,A -95.1986,B 22.9989,C -1.0812,E1 23.0165,E2 542.0375} C_DIS
LIN {X -3.0301,Y -123.4918,Z 141,A -93.728,B 22.9988,C -1.0841,E1 23.0206,E2 540.5592} C_DIS
LIN {X -0.0042,Y -123.5302,Z 141,A -92.2793,B 22.9987,C -1.0863,E1 23.0247,E2 539.1048} C_DIS
LIN {X -0.0042,Y -123.5302,Z 141,A -92.2793,B 22.9987,C -1.0863,E1 23.0247,E2 539.1048} C_DIS
Enddeposition()
LIN {X 0.9125,Y -128.7852,Z 142,A -92.8338,B 24.9658,C -1.3518,E1 25.0013,E2 539.2712} C_DIS
Startdeposition()
$VEL.CP = VEL_PRINT
LIN {X 4.949,Y -128.6939,Z 142,A -90.6772,B 24.9648,C -1.3707,E1 25.0075,E2 537.0703} C_DIS
LIN {X 8.6468,Y -128.5004,Z 142,A -88.9424,B 24.9645,C -1.3758,E1 25.0124,E2 535.324} C_DIS
LIN {X 12.2588,Y -128.2042,Z 142,A -87.5197,B 24.965,C -1.367,E1 25.0163,E2 533.923} C_DIS
LIN {X 14.6388,Y -127.9557,Z 142,A -86.4368,B 24.965,C -1.3685,E1 25.0193,E2 532.8373} C_DIS
LIN {X 17.8725,Y -127.5432,Z 142,A -85.0085,B 24.965,C -1.3684,E1 25.0232,E2 531.4104} C_DIS
LIN {X 20.5736,Y -127.1365,Z 142,A -83.5874,B 24.9643,C -1.3799,E1 25.0272,E2 529.9636} C_DIS
LIN {X 24.0678,Y -126.52,Z 142,A -82.1446,B 24.9646,C -1.3742,E1 25.0311,E2 528.5358} C_DIS
LIN {X 26.7638,Y -125.9778,Z 142,A -80.8901,B 24.9645,C -1.3769,E1 25.0346,E2 527.2765} C_DIS
LIN {X 29.8231,Y -125.2887,Z 142,A -79.6453,B 24.9648,C -1.3705,E1 25.0379,E2 526.0485} C_DIS
LIN {X 32.8513,Y -124.5288,Z 142,A -78.1913,B 24.9646,C -1.3753,E1 25.0419,E2 524.5855} C_DIS
LIN {X 35.7634,Y -123.7243,Z 142,A -76.7237,B 24.9642,C -1.3832,E1 25.0459,E2 523.1015} C_DIS
LIN {X 38.4406,Y -122.9205,Z 142,A -75.4435,B 24.964,C -1.3865,E1 25.0493,E2 521.8157} C_DIS
LIN {X 41.8429,Y -121.8023,Z 142,A -74.0709,B 24.9645,C -1.3771,E1 25.0529,E2 520.4681} C_DIS
LIN {X 44.7691,Y -120.7576,Z 142,A -72.5244,B 24.9639,C -1.3875,E1 25.057,E2 518.9001} C_DIS
LIN {X 47.9282,Y -119.5384,Z 142,A -71.0772,B 24.9639,C -1.3866,E1 25.0607,E2 517.4584} C_DIS
LIN {X 50.3724,Y -118.5316,Z 142,A -69.7913,B 24.9636,C -1.3941,E1 25.0641,E2 516.1579} C_DIS
LIN {X 53.4419,Y -117.1789,Z 142,A -68.3565,B 24.9636,C -1.3934,E1 25.0677,E2 514.7283} C_DIS
LIN {X 56.5259,Y -115.7219,Z 142,A -66.9643,B 24.9638,C -1.3893,E1 25.0712,E2 513.3493} C_DIS
LIN {X 59.2725,Y -114.3403,Z 142,A -65.4297,B 24.9633,C -1.4004,E1 25.075,E2 511.7928} C_DIS
LIN {X 62.8053,Y -112.4392,Z 142,A -63.7579,B 24.9634,C -1.3976,E1 25.0791,E2 510.1323} C_DIS
LIN {X 66.2361,Y -110.453,Z 142,A -61.975,B 24.9632,C -1.402,E1 25.0834,E2 508.3447} C_DIS
LIN {X 69.3028,Y -108.5546,Z 142,A -60.3008,B 24.9628,C -1.4088,E1 25.0874,E2 506.6597} C_DIS
LIN {X 72.6524,Y -106.3422,Z 142,A -58.4945,B 24.9626,C -1.4135,E1 25.0916,E2 504.8484} C_DIS
LIN {X 76.441,Y -103.6522,Z 142,A -56.5263,B 24.9626,C -1.4126,E1 25.096,E2 502.8891} C_DIS
LIN {X 79.2806,Y -101.4971,Z 142,A -54.8502,B 24.9622,C -1.4209,E1 25.0998,E2 501.1996} C_DIS
LIN {X 82.7183,Y -98.715,Z 142,A -52.942,B 24.9622,C -1.4222,E1 25.1039,E2 499.2956} C_DIS
LIN {X 85.8349,Y -96.0174,Z 142,A -51.1078,B 24.9619,C -1.4265,E1 25.1077,E2 497.4585} C_DIS
LIN {X 88.7312,Y -93.348,Z 142,A -49.4362,B 24.9619,C -1.4265,E1 25.1111,E2 495.7939} C_DIS
LIN {X 91.6078,Y -90.5267,Z 142,A -47.6251,B 24.9616,C -1.4319,E1 25.1147,E2 493.9776} C_DIS
LIN {X 94.4884,Y -87.5158,Z 142,A -45.8016,B 24.9614,C -1.4351,E1 25.1182,E2 492.1546} C_DIS
LIN {X 96.8907,Y -84.8481,Z 142,A -44.1247,B 24.961,C -1.4435,E1 25.1213,E2 490.4652} C_DIS
LIN {X 99.8465,Y -81.3491,Z 142,A -42.1781,B 24.961,C -1.4441,E1 25.1248,E2 488.5262} C_DIS
LIN {X 102.1832,Y -78.3937,Z 142,A -40.4415,B 24.9605,C -1.4519,E1 25.1278,E2 486.7793} C_DIS
LIN {X 104.5639,Y -75.1895,Z 142,A -38.6486,B 24.9602,C -1.4578,E1 25.1307,E2 484.9813} C_DIS
LIN {X 106.9484,Y -71.7571,Z 142,A -36.8131,B 24.96,C -1.4618,E1 25.1336,E2 483.1453} C_DIS
LIN {X 109.166,Y -68.3363,Z 142,A -34.9954,B 24.9597,C -1.4673,E1 25.1363,E2 481.3238} C_DIS
LIN {X 111.3527,Y -64.7115,Z 142,A -33.1531,B 24.9595,C -1.4707,E1 25.139,E2 479.4831} C_DIS
LIN {X 113.508,Y -60.8515,Z 142,A -31.1777,B 24.9591,C -1.4771,E1 25.1416,E2 477.5031} C_DIS
LIN {X 115.2757,Y -57.4302,Z 142,A -29.6903,B 24.9595,C -1.4701,E1 25.1435,E2 476.0398} C_DIS
LIN {X 116.5568,Y -54.7871,Z 142,A -28.1898,B 24.9587,C -1.4846,E1 25.1453,E2 474.5135} C_DIS
LIN {X 118.0555,Y -51.4737,Z 142,A -26.6771,B 24.9587,C -1.4839,E1 25.147,E2 473.0104} C_DIS
LIN {X 119.3487,Y -48.3989,Z 142,A -25.2545,B 24.9587,C -1.4853,E1 25.1485,E2 471.5924} C_DIS
LIN {X 120.5265,Y -45.3862,Z 142,A -23.9615,B 24.9589,C -1.482,E1 25.1498,E2 470.3145} C_DIS
LIN {X 121.6077,Y -42.4044,Z 142,A -22.57,B 24.9587,C -1.4854,E1 25.1511,E2 468.9226} C_DIS
LIN {X 122.6047,Y -39.4292,Z 142,A -21.0426,B 24.958,C -1.4969,E1 25.1524,E2 467.3767} C_DIS
LIN {X 123.4748,Y -36.6155,Z 142,A -19.7132,B 24.9577,C -1.5022,E1 25.1535,E2 466.0426} C_DIS
LIN {X 124.3121,Y -33.6641,Z 142,A -18.2876,B 24.9573,C -1.5099,E1 25.1546,E2 464.607} C_DIS
LIN {X 125.0781,Y -30.6965,Z 142,A -16.9288,B 24.9571,C -1.5141,E1 25.1555,E2 463.2462} C_DIS
LIN {X 125.8336,Y -27.4321,Z 142,A -15.6741,B 24.9575,C -1.5062,E1 25.1563,E2 462.0173} C_DIS
LIN {X 126.4527,Y -24.4196,Z 142,A -14.2596,B 24.9571,C -1.5132,E1 25.157,E2 460.5946} C_DIS
LIN {X 126.9082,Y -21.9414,Z 142,A -13.0268,B 24.9566,C -1.5229,E1 25.1577,E2 459.3463} C_DIS
LIN {X 127.3875,Y -18.9617,Z 142,A -11.696,B 24.9563,C -1.5266,E1 25.1582,E2 458.0144} C_DIS
LIN {X 127.794,Y -15.9945,Z 142,A -10.3756,B 24.9561,C -1.5304,E1 25.1587,E2 456.6929} C_DIS
LIN {X 128.1289,Y -13.0423,Z 142,A -8.9414,B 24.9555,C -1.5408,E1 25.1591,E2 455.2426} C_DIS
LIN {X 128.3938,Y -10.1072,Z 142,A -7.7666,B 24.9557,C -1.5378,E1 25.1594,E2 454.082} C_DIS
LIN {X 128.6171,Y -6.6546,Z 142,A -6.3276,B 24.9557,C -1.5375,E1 25.1596,E2 452.6522} C_DIS
LIN {X 128.7396,Y -3.5655,Z 142,A -4.8518,B 24.9551,C -1.5475,E1 25.1598,E2 451.1617} C_DIS
LIN {X 128.789,Y 0.5129,Z 142,A -3.1449,B 24.9551,C -1.5476,E1 25.1598,E2 449.4646} C_DIS
LIN {X 128.756,Y 2.9778,Z 142,A -2.0771,B 24.9551,C -1.5497,E1 25.1598,E2 448.3982} C_DIS
LIN {X 128.6569,Y 5.8616,Z 142,A -0.6113,B 24.9542,C -1.5637,E1 25.1596,E2 446.9081} C_DIS
LIN {X 128.4916,Y 8.7678,Z 142,A 0.5363,B 24.9544,C -1.56,E1 25.1594,E2 445.776} C_DIS
LIN {X 128.2584,Y 11.6942,Z 142,A 1.9743,B 24.9537,C -1.5714,E1 25.159,E2 444.3197} C_DIS
LIN {X 127.8663,Y 15.3882,Z 142,A 3.54,B 24.9537,C -1.5721,E1 25.1585,E2 442.7616} C_DIS
LIN {X 127.3529,Y 19.1855,Z 142,A 5.2275,B 24.9534,C -1.5767,E1 25.1578,E2 441.0733} C_DIS
LIN {X 126.832,Y 22.3673,Z 142,A 6.6495,B 24.9532,C -1.5806,E1 25.1572,E2 439.6503} C_DIS
LIN {X 126.199,Y 25.6976,Z 142,A 8.1201,B 24.953,C -1.5834,E1 25.1564,E2 438.1817} C_DIS
LIN {X 125.5411,Y 28.7399,Z 142,A 9.4073,B 24.953,C -1.5826,E1 25.1556,E2 436.904} C_DIS
LIN {X 124.8773,Y 31.4995,Z 142,A 10.7208,B 24.9527,C -1.5893,E1 25.1547,E2 435.5823} C_DIS
LIN {X 124.0817,Y 34.5006,Z 142,A 12.0034,B 24.9527,C -1.5883,E1 25.1538,E2 434.3093} C_DIS
LIN {X 123.3418,Y 37.064,Z 142,A 13.4165,B 24.9518,C -1.6041,E1 25.1526,E2 432.8671} C_DIS
LIN {X 122.2446,Y 40.5314,Z 142,A 14.8025,B 24.9522,C -1.5967,E1 25.1515,E2 431.5064} C_DIS
LIN {X 121.2543,Y 43.4049,Z 142,A 16.2385,B 24.9517,C -1.6052,E1 25.1501,E2 430.0583} C_DIS
LIN {X 120.1667,Y 46.3313,Z 142,A 17.5047,B 24.9519,C -1.6029,E1 25.1489,E2 428.8048} C_DIS
LIN {X 119.15,Y 48.8918,Z 142,A 19.0038,B 24.9508,C -1.6211,E1 25.1473,E2 427.271} C_DIS
LIN {X 117.6356,Y 52.4249,Z 142,A 20.5579,B 24.951,C -1.6178,E1 25.1456,E2 425.7331} C_DIS
LIN {X 116.3218,Y 55.2792,Z 142,A 21.7249,B 24.9515,C -1.6096,E1 25.1442,E2 424.5918} C_DIS
LIN {X 114.949,Y 58.0804,Z 142,A 23.3617,B 24.9504,C -1.6268,E1 25.1422,E2 422.9232} C_DIS
LIN {X 113.2594,Y 61.3143,Z 142,A 25.0549,B 24.9499,C -1.635,E1 25.1399,E2 421.2194} C_DIS
LIN {X 111.2035,Y 64.9679,Z 142,A 26.919,B 24.9496,C -1.6401,E1 25.1373,E2 419.3529} C_DIS
LIN {X 109.0133,Y 68.5792,Z 142,A 28.7719,B 24.9494,C -1.6438,E1 25.1346,E2 417.5008} C_DIS
LIN {X 106.6042,Y 72.267,Z 142,A 30.6929,B 24.9492,C -1.6469,E1 25.1316,E2 415.5821} C_DIS
LIN {X 104.2025,Y 75.6889,Z 142,A 32.5386,B 24.9489,C -1.6509,E1 25.1286,E2 413.7359} C_DIS
LIN {X 101.7147,Y 79.0006,Z 142,A 34.3565,B 24.9487,C -1.6542,E1 25.1255,E2 411.9188} C_DIS
LIN {X 99.1991,Y 82.1371,Z 142,A 36.1625,B 24.9484,C -1.6594,E1 25.1224,E2 410.1088} C_DIS
LIN {X 96.2913,Y 85.528,Z 142,A 38.1154,B 24.9482,C -1.6623,E1 25.1188,E2 408.158} C_DIS
LIN {X 93.3957,Y 88.6813,Z 142,A 40.0632,B 24.9478,C -1.6689,E1 25.115,E2 406.2032} C_DIS
LIN {X 90.3939,Y 91.7387,Z 142,A 41.973,B 24.9475,C -1.6732,E1 25.1113,E2 404.2911} C_DIS
LIN {X 87.2174,Y 94.7633,Z 142,A 43.873,B 24.9475,C -1.6746,E1 25.1074,E2 402.3956} C_DIS
LIN {X 83.8787,Y 97.7311,Z 142,A 45.7936,B 24.9475,C -1.6752,E1 25.1034,E2 400.4814} C_DIS
LIN {X 80.6622,Y 100.4023,Z 142,A 47.7198,B 24.947,C -1.6822,E1 25.0992,E2 398.5459} C_DIS
LIN {X 77.2489,Y 103.0521,Z 142,A 49.6624,B 24.9467,C -1.6868,E1 25.0949,E2 396.5996} C_DIS
LIN {X 73.75,Y 105.5838,Z 142,A 51.5669,B 24.9465,C -1.6892,E1 25.0905,E2 394.6958} C_DIS
LIN {X 70.0454,Y 108.0768,Z 142,A 53.4915,B 24.9465,C -1.6893,E1 25.0861,E2 392.7774} C_DIS
LIN {X 66.5063,Y 110.2901,Z 142,A 55.361,B 24.9463,C -1.6928,E1 25.0816,E2 390.9055} C_DIS
LIN {X 62.7462,Y 112.4724,Z 142,A 57.3065,B 24.9461,C -1.6962,E1 25.0769,E2 388.9578} C_DIS
LIN {X 59.1293,Y 114.4151,Z 142,A 59.0788,B 24.9461,C -1.6959,E1 25.0725,E2 387.1912} C_DIS
LIN {X 55.798,Y 116.0739,Z 142,A 60.475,B 24.9468,C -1.6848,E1 25.0691,E2 385.8251} C_DIS
LIN {X 53.3205,Y 117.235,Z 142,A 61.9346,B 24.9459,C -1.6986,E1 25.0653,E2 384.3366} C_DIS
LIN {X 49.9814,Y 118.6949,Z 142,A 63.4182,B 24.9463,C -1.6934,E1 25.0616,E2 382.8687} C_DIS
LIN {X 46.9339,Y 119.9324,Z 142,A 64.9699,B 24.9459,C -1.6994,E1 25.0575,E2 381.3063} C_DIS
LIN {X 43.9056,Y 121.0737,Z 142,A 66.2835,B 24.9462,C -1.6944,E1 25.0541,E2 380.0073} C_DIS
LIN {X 41.2281,Y 122.0126,Z 142,A 67.7043,B 24.9456,C -1.7035,E1 25.0503,E2 378.5678} C_DIS
LIN {X 38.0013,Y 123.0549,Z 142,A 69.1381,B 24.9458,C -1.701,E1 25.0465,E2 377.1426} C_DIS
LIN {X 35.3884,Y 123.8334,Z 142,A 70.474,B 24.9453,C -1.708,E1 25.0429,E2 375.7922} C_DIS
LIN {X 32.3088,Y 124.6719,Z 142,A 71.8656,B 24.9453,C -1.7075,E1 25.0391,E2 374.404} C_DIS
LIN {X 29.3642,Y 125.3984,Z 142,A 73.2376,B 24.9453,C -1.7095,E1 25.0354,E2 373.0294} C_DIS
LIN {X 25.9602,Y 126.1455,Z 142,A 74.7257,B 24.9453,C -1.7071,E1 25.0314,E2 371.5489} C_DIS
LIN {X 22.7746,Y 126.7591,Z 142,A 76.1468,B 24.9454,C -1.7066,E1 25.0275,E2 370.1305} C_DIS
LIN {X 19.5953,Y 127.2894,Z 142,A 77.5742,B 24.9454,C -1.7067,E1 25.0235,E2 368.7043} C_DIS
LIN {X 15.6732,Y 127.8323,Z 142,A 79.3217,B 24.9454,C -1.7064,E1 25.0187,E2 366.9589} C_DIS
LIN {X 11.515,Y 128.2749,Z 142,A 81.1364,B 24.9456,C -1.7043,E1 25.0137,E2 365.1502} C_DIS
LIN {X 8.5263,Y 128.5079,Z 142,A 82.4423,B 24.9456,C -1.703,E1 25.01,E2 363.8481} C_DIS
LIN {X 5.6219,Y 128.6676,Z 142,A 83.734,B 24.9456,C -1.7029,E1 25.0064,E2 362.5572} C_DIS
LIN {X 2.8586,Y 128.7593,Z 142,A 85.1706,B 24.945,C -1.713,E1 25.0024,E2 361.0969} C_DIS
LIN {X -0.8891,Y 128.7861,Z 142,A 86.7777,B 24.9452,C -1.7097,E1 24.9979,E2 359.4977} C_DIS
LIN {X -4.3657,Y 128.7166,Z 142,A 88.2475,B 24.9455,C -1.7054,E1 24.9938,E2 358.0378} C_DIS
LIN {X -7.1915,Y 128.5901,Z 142,A 89.5348,B 24.9455,C -1.7064,E1 24.9902,E2 356.7478} C_DIS
LIN {X -10.5421,Y 128.3571,Z 142,A 91.0179,B 24.9455,C -1.7052,E1 24.9861,E2 355.267} C_DIS
LIN {X -13.836,Y 128.0435,Z 142,A 92.512,B 24.9455,C -1.7055,E1 24.982,E2 353.7712} C_DIS
LIN {X -17.8386,Y 127.548,Z 142,A 94.2794,B 24.9456,C -1.7031,E1 24.9771,E2 352.0084} C_DIS
LIN {X -20.5962,Y 127.1327,Z 142,A 95.6358,B 24.9453,C -1.7079,E1 24.9733,E2 350.6394} C_DIS
LIN {X -23.7697,Y 126.577,Z 142,A 96.9534,B 24.9458,C -1.7011,E1 24.9697,E2 349.3366} C_DIS
LIN {X -26.8637,Y 125.9563,Z 142,A 98.3355,B 24.9459,C -1.6988,E1 24.9659,E2 347.9582} C_DIS
LIN {X -30.0099,Y 125.2436,Z 142,A 99.788,B 24.9459,C -1.6983,E1 24.962,E2 346.5049} C_DIS
LIN {X -32.9798,Y 124.4946,Z 142,A 101.1254,B 24.9461,C -1.6957,E1 24.9584,E2 345.1718} C_DIS
LIN {X -35.8297,Y 123.7048,Z 142,A 102.3848,B 24.9464,C -1.6915,E1 24.955,E2 343.9202} C_DIS
LIN {X -38.6304,Y 122.8598,Z 142,A 103.8654,B 24.9459,C -1.6987,E1 24.951,E2 342.42} C_DIS
LIN {X -41.4383,Y 121.9426,Z 142,A 105.1105,B 24.9462,C -1.6937,E1 24.9478,E2 341.1844} C_DIS
LIN {X -44.5517,Y 120.839,Z 142,A 106.5331,B 24.9465,C -1.6896,E1 24.944,E2 339.7689} C_DIS
LIN {X -47.4073,Y 119.7484,Z 142,A 108.0769,B 24.9461,C -1.6966,E1 24.94,E2 338.2052} C_DIS
LIN {X -50.8679,Y 118.3174,Z 142,A 109.6302,B 24.9466,C -1.6887,E1 24.936,E2 336.6669} C_DIS
LIN {X -53.7148,Y 117.0527,Z 142,A 110.9084,B 24.947,C -1.6814,E1 24.9328,E2 335.403} C_DIS
LIN {X -56.7321,Y 115.6201,Z 142,A 112.5006,B 24.9468,C -1.6842,E1 24.9288,E2 333.8002} C_DIS
LIN {X -59.454,Y 114.245,Z 142,A 113.9292,B 24.9468,C -1.6853,E1 24.9252,E2 332.3648} C_DIS
LIN {X -63.189,Y 112.2236,Z 142,A 115.8155,B 24.947,C -1.6818,E1 24.9206,E2 330.4815} C_DIS
LIN {X -66.6993,Y 110.1733,Z 142,A 117.6584,B 24.9471,C -1.6801,E1 24.9162,E2 328.637} C_DIS
LIN {X -69.8415,Y 108.2092,Z 142,A 119.243,B 24.9475,C -1.6739,E1 24.9125,E2 327.0622} C_DIS
LIN {X -72.5918,Y 106.3838,Z 142,A 120.8565,B 24.9472,C -1.6779,E1 24.9087,E2 325.4338} C_DIS
LIN {X -75.916,Y 104.0379,Z 142,A 122.6731,B 24.9475,C -1.6744,E1 24.9046,E2 323.6192} C_DIS
LIN {X -79.2806,Y 101.4971,Z 142,A 124.4227,B 24.9481,C -1.6644,E1 24.9007,E2 321.8871} C_DIS
LIN {X -81.8736,Y 99.4172,Z 142,A 125.9964,B 24.9481,C -1.6656,E1 24.8973,E2 320.3045} C_DIS
LIN {X -85.0438,Y 96.7193,Z 142,A 127.9088,B 24.9481,C -1.6642,E1 24.8933,E2 318.388} C_DIS
LIN {X -88.0751,Y 93.9676,Z 142,A 129.6013,B 24.9488,C -1.6537,E1 24.8898,E2 316.7135} C_DIS
LIN {X -90.5267,Y 91.6078,Z 142,A 131.262,B 24.9485,C -1.657,E1 24.8865,E2 315.038} C_DIS
LIN {X -93.5747,Y 88.4916,Z 142,A 133.1737,B 24.9489,C -1.6508,E1 24.8828,E2 313.1327} C_DIS
LIN {X -96.6103,Y 85.1671,Z 142,A 135.1184,B 24.9494,C -1.6429,E1 24.8792,E2 311.1982} C_DIS
LIN {X -98.9307,Y 82.4611,Z 142,A 136.6807,B 24.9497,C -1.6376,E1 24.8764,E2 309.6415} C_DIS
LIN {X -101.0771,Y 79.8153,Z 142,A 138.3314,B 24.9497,C -1.6399,E1 24.8735,E2 307.9776} C_DIS
LIN {X -103.6569,Y 76.4347,Z 142,A 140.225,B 24.9499,C -1.6348,E1 24.8703,E2 306.0871} C_DIS
LIN {X -106.2233,Y 72.8256,Z 142,A 142.1413,B 24.9504,C -1.6267,E1 24.8673,E2 304.1805} C_DIS
LIN {X -108.5195,Y 69.3577,Z 142,A 143.9953,B 24.9507,C -1.6216,E1 24.8645,E2 302.3294} C_DIS
LIN {X -110.5656,Y 66.0472,Z 142,A 145.7824,B 24.9509,C -1.6191,E1 24.8619,E2 300.539} C_DIS
LIN {X -112.7441,Y 62.2555,Z 142,A 147.7299,B 24.9512,C -1.6135,E1 24.8592,E2 298.5948} C_DIS
LIN {X -114.6321,Y 58.7029,Z 142,A 149.4038,B 24.9519,C -1.6027,E1 24.857,E2 296.9376} C_DIS
LIN {X -115.9056,Y 56.1503,Z 142,A 150.8345,B 24.9517,C -1.6064,E1 24.8553,E2 295.4905} C_DIS
LIN {X -117.235,Y 53.3205,Z 142,A 152.2522,B 24.9518,C -1.6033,E1 24.8536,E2 294.0723} C_DIS
LIN {X -118.5828,Y 50.2498,Z 142,A 153.671,B 24.9523,C -1.5953,E1 24.8521,E2 292.6647} C_DIS
LIN {X -119.9447,Y 46.9022,Z 142,A 155.2633,B 24.9527,C -1.5896,E1 24.8504,E2 291.0772} C_DIS
LIN {X -120.9299,Y 44.3045,Z 142,A 156.4797,B 24.9529,C -1.5847,E1 24.8493,E2 289.8655} C_DIS
LIN {X -121.9426,Y 41.4383,Z 142,A 157.8881,B 24.953,C -1.583,E1 24.848,E2 288.4531} C_DIS
LIN {X -122.9829,Y 38.2367,Z 142,A 159.3546,B 24.9534,C -1.5768,E1 24.8467,E2 286.993} C_DIS
LIN {X -123.9026,Y 35.1408,Z 142,A 160.7979,B 24.9537,C -1.5725,E1 24.8456,E2 285.5516} C_DIS
LIN {X -124.7276,Y 32.0895,Z 142,A 162.0624,B 24.9543,C -1.5614,E1 24.8447,E2 284.3063} C_DIS
LIN {X -125.3836,Y 29.4294,Z 142,A 163.532,B 24.9539,C -1.569,E1 24.8437,E2 282.8098} C_DIS
LIN {X -126.1008,Y 26.1799,Z 142,A 165.0132,B 24.9542,C -1.5643,E1 24.8429,E2 281.3312} C_DIS
LIN {X -126.6912,Y 23.1541,Z 142,A 166.3902,B 24.9544,C -1.56,E1 24.8422,E2 279.9562} C_DIS
LIN {X -127.2076,Y 20.1235,Z 142,A 167.555,B 24.9552,C -1.5461,E1 24.8417,E2 278.8176} C_DIS
LIN {X -127.6528,Y 17.0714,Z 142,A 168.9516,B 24.9554,C -1.5428,E1 24.8411,E2 277.4208} C_DIS
LIN {X -128.0237,Y 14.0206,Z 142,A 170.4408,B 24.9554,C -1.5439,E1 24.8406,E2 275.9198} C_DIS
LIN {X -128.3321,Y 10.838,Z 142,A 171.868,B 24.9556,C -1.5395,E1 24.8403,E2 274.4947} C_DIS
LIN {X -128.5786,Y 7.3773,Z 142,A 173.4595,B 24.9558,C -1.5366,E1 24.84,E2 272.9005} C_DIS
LIN {X -128.7305,Y 3.8947,Z 142,A 175,B 24.9561,C -1.531,E1 24.8398,E2 271.364} C_DIS
LIN {X -128.7893,Y 0.477,Z 142,A 176.6073,B 24.9561,C -1.53,E1 24.8398,E2 269.7493} C_DIS
LIN {X -128.756,Y -2.9778,Z 142,A 178.162,B 24.9564,C -1.5258,E1 24.8398,E2 268.1953} C_DIS
LIN {X -128.645,Y -6.0981,Z 142,A 179.4894,B 24.9568,C -1.5184,E1 24.84,E2 266.8776} C_DIS
LIN {X -128.4583,Y -9.2243,Z 142,A -179.0952,B 24.957,C -1.5149,E1 24.8403,E2 265.4621} C_DIS
LIN {X -128.1802,Y -12.5083,Z 142,A -177.5669,B 24.9571,C -1.513,E1 24.8407,E2 263.929} C_DIS
LIN {X -127.7168,Y -16.5838,Z 142,A -175.904,B 24.9579,C -1.4995,E1 24.8412,E2 262.2883} C_DIS
LIN {X -127.3781,Y -19.0223,Z 142,A -174.6,B 24.9575,C -1.5057,E1 24.8418,E2 260.9618} C_DIS
LIN {X -126.8042,Y -22.5227,Z 142,A -173.2347,B 24.9584,C -1.4908,E1 24.8424,E2 259.624} C_DIS
LIN {X -126.3549,Y -24.9312,Z 142,A -171.8737,B 24.9579,C -1.4999,E1 24.8431,E2 258.2332} C_DIS
LIN {X -125.5746,Y -28.5932,Z 142,A -170.412,B 24.9587,C -1.4851,E1 24.844,E2 256.7981} C_DIS
LIN {X -124.8807,Y -31.4862,Z 142,A -168.9895,B 24.9587,C -1.4856,E1 24.8449,E2 255.3662} C_DIS
LIN {X -124.1148,Y -34.3823,Z 142,A -167.6354,B 24.9588,C -1.4824,E1 24.8459,E2 254.0118} C_DIS
LIN {X -123.3288,Y -37.1066,Z 142,A -166.3376,B 24.959,C -1.4802,E1 24.847,E2 252.7117} C_DIS
LIN {X -122.4001,Y -40.0643,Z 142,A -164.9016,B 24.959,C -1.4787,E1 24.8482,E2 251.2712} C_DIS
LIN {X -121.2073,Y -43.5351,Z 142,A -163.5454,B 24.96,C -1.4608,E1 24.8494,E2 249.95} C_DIS
LIN {X -120.1784,Y -46.301,Z 142,A -162.0575,B 24.9598,C -1.465,E1 24.8509,E2 248.4435} C_DIS
LIN {X -118.9841,Y -49.2889,Z 142,A -160.6214,B 24.96,C -1.461,E1 24.8524,E2 247.009} C_DIS
LIN {X -117.7767,Y -52.1094,Z 142,A -159.1575,B 24.96,C -1.4617,E1 24.8541,E2 245.5354} C_DIS
LIN {X -116.499,Y -54.9082,Z 142,A -157.8346,B 24.9603,C -1.4555,E1 24.8556,E2 244.22} C_DIS
LIN {X -114.9544,Y -58.0699,Z 142,A -156.2275,B 24.9604,C -1.4531,E1 24.8576,E2 242.6101} C_DIS
LIN {X -113.2594,Y -61.3143,Z 142,A -154.5951,B 24.9607,C -1.4487,E1 24.8598,E2 240.9795} C_DIS
LIN {X -111.2553,Y -64.8798,Z 142,A -152.7349,B 24.9609,C -1.4456,E1 24.8623,E2 239.1169} C_DIS
LIN {X -109.1073,Y -68.4301,Z 142,A -150.8366,B 24.9609,C -1.4431,E1 24.8651,E2 237.2149} C_DIS
LIN {X -106.8855,Y -71.8513,Z 142,A -148.9766,B 24.9611,C -1.4405,E1 24.868,E2 235.3517} C_DIS
LIN {X -104.3495,Y -75.4861,Z 142,A -147.0415,B 24.9615,C -1.4337,E1 24.8711,E2 233.4232} C_DIS
LIN {X -101.8771,Y -78.7911,Z 142,A -145.1903,B 24.9617,C -1.4299,E1 24.8743,E2 231.5724} C_DIS
LIN {X -99.3199,Y -81.9911,Z 142,A -143.3441,B 24.9619,C -1.4266,E1 24.8775,E2 229.7253} C_DIS
LIN {X -96.4849,Y -85.309,Z 142,A -141.4186,B 24.9622,C -1.4213,E1 24.881,E2 227.8037} C_DIS
LIN {X -93.4431,Y -88.6311,Z 142,A -139.3712,B 24.9622,C -1.4189,E1 24.8849,E2 225.7532} C_DIS
LIN {X -90.4777,Y -91.6565,Z 142,A -137.5833,B 24.9628,C -1.4102,E1 24.8884,E2 223.9784} C_DIS
LIN {X -87.8558,Y -94.1718,Z 142,A -135.8797,B 24.9628,C -1.411,E1 24.8919,E2 222.266} C_DIS
LIN {X -84.5879,Y -97.1178,Z 142,A -133.9435,B 24.963,C -1.406,E1 24.896,E2 220.3339} C_DIS
LIN {X -81.2301,Y -99.9437,Z 142,A -131.9997,B 24.9632,C -1.4018,E1 24.9001,E2 218.3926} C_DIS
LIN {X -78.2193,Y -102.3166,Z 142,A -130.255,B 24.9632,C -1.4006,E1 24.904,E2 216.6444} C_DIS
LIN {X -74.764,Y -104.8682,Z 142,A -128.353,B 24.9635,C -1.3968,E1 24.9083,E2 214.7447} C_DIS
LIN {X -71.1934,Y -107.3248,Z 142,A -126.3809,B 24.9635,C -1.3958,E1 24.9128,E2 212.7686} C_DIS
LIN {X -67.6957,Y -109.5647,Z 142,A -124.5031,B 24.9635,C -1.3944,E1 24.9173,E2 210.8882} C_DIS
LIN {X -64.0989,Y -111.7068,Z 142,A -122.689,B 24.9638,C -1.3893,E1 24.9217,E2 209.0807} C_DIS
LIN {X -60.5956,Y -113.6455,Z 142,A -120.8514,B 24.9638,C -1.3896,E1 24.9262,E2 207.2372} C_DIS
LIN {X -57.3258,Y -115.3273,Z 142,A -119.3337,B 24.9642,C -1.3817,E1 24.9299,E2 205.7341} C_DIS
LIN {X -54.4977,Y -116.6907,Z 142,A -117.8725,B 24.9642,C -1.3832,E1 24.9336,E2 204.2656} C_DIS
LIN {X -51.7265,Y -117.9462,Z 142,A -116.5111,B 24.9642,C -1.3821,E1 24.9371,E2 202.9037} C_DIS
LIN {X -48.5345,Y -119.294,Z 142,A -114.9863,B 24.9643,C -1.3797,E1 24.941,E2 201.3812} C_DIS
LIN {X -45.3907,Y -120.5248,Z 142,A -113.6579,B 24.9649,C -1.3696,E1 24.9444,E2 200.0738} C_DIS
LIN {X -42.8106,Y -121.4668,Z 142,A -112.2281,B 24.9644,C -1.3788,E1 24.9483,E2 198.6193} C_DIS
LIN {X -39.8161,Y -122.4811,Z 142,A -110.8228,B 24.9644,C -1.3776,E1 24.952,E2 197.2143} C_DIS
LIN {X -36.7378,Y -123.439,Z 142,A -109.4163,B 24.9646,C -1.3752,E1 24.9558,E2 195.8111} C_DIS
LIN {X -33.612,Y -124.326,Z 142,A -108.0076,B 24.9647,C -1.3724,E1 24.9595,E2 194.4069} C_DIS
LIN {X -30.5865,Y -125.1046,Z 142,A -106.5702,B 24.9647,C -1.374,E1 24.9634,E2 192.9637} C_DIS
LIN {X -27.6749,Y -125.7811,Z 142,A -105.3584,B 24.965,C -1.3674,E1 24.9667,E2 191.766} C_DIS
LIN {X -24.8073,Y -126.3786,Z 142,A -104.0083,B 24.9649,C -1.3692,E1 24.9704,E2 190.41} C_DIS
LIN {X -21.9414,Y -126.9082,Z 142,A -102.667,B 24.9648,C -1.371,E1 24.9741,E2 189.0631} C_DIS
LIN {X -18.9617,Y -127.3875,Z 142,A -101.3261,B 24.9648,C -1.3705,E1 24.9778,E2 187.7221} C_DIS
LIN {X -15.3817,Y -127.8671,Z 142,A -99.9387,B 24.9654,C -1.3592,E1 24.9816,E2 186.3606} C_DIS
LIN {X -12.4596,Y -128.1849,Z 142,A -98.4807,B 24.965,C -1.3666,E1 24.9857,E2 184.8841} C_DIS
LIN {X -8.5263,Y -128.5079,Z 142,A -96.5669,B 24.9646,C -1.3746,E1 24.9911,E2 182.9506} C_DIS
LIN {X -4.8237,Y -128.6988,Z 142,A -95.0075,B 24.9648,C -1.3702,E1 24.9954,E2 181.4014} C_DIS
LIN {X -1.3081,Y -128.7838,Z 142,A -93.5488,B 24.9651,C -1.3651,E1 24.9994,E2 179.9548} C_DIS
LIN {X 0.9125,Y -128.7852,Z 142,A -92.8332,B 24.9658,C -1.3515,E1 25.0014,E2 179.2712} C_DIS
Enddeposition()
LIN {X 0.9125,Y -128.7852,Z 142,A -92.8332,B 24.9658,C -1.3515,E1 25.0014,E2 179.2712} C_DIS
Startdeposition()
$VEL.CP = VEL_PRINT
LIN {X -2.3484,Y -127.7984,Z 142,A -94.5291,B 24.9655,C -1.3565,E1 24.9966,E2 180.9553} C_DIS
LIN {X -5.0754,Y -127.719,Z 142,A -96.2606,B 24.9668,C -1.3312,E1 24.9916,E2 182.7471} C_DIS
LIN {X -8.8411,Y -127.5145,Z 142,A -97.392,B 24.9654,C -1.3588,E1 24.9887,E2 183.8135} C_DIS
LIN {X -13.5282,Y -127.1019,Z 142,A -99.6601,B 24.9658,C -1.351,E1 24.9823,E2 186.1011} C_DIS
LIN {X -16.7011,Y -126.7239,Z 142,A -101.1242,B 24.9658,C -1.3497,E1 24.9782,E2 187.5694} C_DIS
LIN {X -20.3706,Y -126.1877,Z 142,A -102.8665,B 24.9661,C -1.3462,E1 24.9734,E2 189.3215} C_DIS
LIN {X -24.4724,Y -125.4559,Z 142,A -104.7426,B 24.9661,C -1.3466,E1 24.9683,E2 191.1988} C_DIS
LIN {X -28.3926,Y -124.6262,Z 142,A -106.4187,B 24.9657,C -1.3533,E1 24.9637,E2 192.861} C_DIS
LIN {X -32.2129,Y -123.696,Z 142,A -108.248,B 24.9658,C -1.351,E1 24.9587,E2 194.6983} C_DIS
LIN {X -35.6382,Y -122.751,Z 142,A -109.8009,B 24.9657,C -1.3541,E1 24.9546,E2 196.2466} C_DIS
LIN {X -38.8448,Y -121.7739,Z 142,A -111.2795,B 24.9655,C -1.3564,E1 24.9506,E2 197.7222} C_DIS
LIN {X -44.2225,Y -119.9274,Z 142,A -113.931,B 24.9657,C -1.3536,E1 24.9436,E2 200.3855} C_DIS
LIN {X -47.6412,Y -118.6091,Z 142,A -115.3302,B 24.965,C -1.367,E1 24.9401,E2 201.7558} C_DIS
LIN {X -52.3353,Y -116.614,Z 142,A -117.7843,B 24.9653,C -1.3614,E1 24.9337,E2 204.2291} C_DIS
LIN {X -56.0149,Y -114.8932,Z 142,A -119.6645,B 24.9653,C -1.3607,E1 24.929,E2 206.1156} C_DIS
LIN {X -58.7026,Y -113.5447,Z 142,A -121.104,B 24.9655,C -1.358,E1 24.9254,E2 207.5654} C_DIS
LIN {X -62.9341,Y -111.255,Z 142,A -123.231,B 24.9652,C -1.3625,E1 24.9202,E2 209.688} C_DIS
LIN {X -66.582,Y -109.1108,Z 142,A -124.8567,B 24.9644,C -1.3782,E1 24.9164,E2 211.2812} C_DIS
LIN {X -69.6301,Y -107.1909,Z 142,A -126.7117,B 24.9649,C -1.3693,E1 24.9119,E2 213.1633} C_DIS
LIN {X -73.2689,Y -104.7379,Z 142,A -128.6417,B 24.9646,C -1.3744,E1 24.9075,E2 215.0878} C_DIS
LIN {X -76.9533,Y -102.061,Z 142,A -130.7131,B 24.9646,C -1.3766,E1 24.9028,E2 217.1614} C_DIS
LIN {X -80.1813,Y -99.545,Z 142,A -132.3539,B 24.9639,C -1.3892,E1 24.8993,E2 218.7783} C_DIS
LIN {X -83.1082,Y -97.1156,Z 142,A -134.3387,B 24.9644,C -1.3792,E1 24.895,E2 220.7943} C_DIS
LIN {X -86.3318,Y -94.2609,Z 142,A -136.2022,B 24.964,C -1.3863,E1 24.8911,E2 222.6484} C_DIS
LIN {X -89.1167,Y -91.6326,Z 142,A -138.0006,B 24.964,C -1.3861,E1 24.8875,E2 224.4548} C_DIS
LIN {X -92.2099,Y -88.5193,Z 142,A -139.968,B 24.9638,C -1.3904,E1 24.8837,E2 226.4204} C_DIS
LIN {X -95.1713,Y -85.3269,Z 142,A -141.8658,B 24.9634,C -1.3974,E1 24.8801,E2 228.31} C_DIS
LIN {X -97.8825,Y -82.2026,Z 142,A -143.7484,B 24.9633,C -1.4004,E1 24.8767,E2 230.1939} C_DIS
LIN {X -100.6439,Y -78.7978,Z 142,A -145.6377,B 24.9628,C -1.4087,E1 24.8734,E2 232.0723} C_DIS
LIN {X -103.372,Y -75.1832,Z 142,A -147.8018,B 24.9628,C -1.4076,E1 24.8698,E2 234.2496} C_DIS
LIN {X -105.4305,Y -72.2679,Z 142,A -149.8284,B 24.9637,C -1.392,E1 24.8665,E2 236.3233} C_DIS
LIN {X -107.8078,Y -68.6717,Z 142,A -151.344,B 24.9624,C -1.4163,E1 24.8643,E2 237.7887} C_DIS
LIN {X -110.0547,Y -65.01,Z 142,A -153.2728,B 24.9622,C -1.4214,E1 24.8615,E2 239.7154} C_DIS
LIN {X -112.1331,Y -61.3552,Z 142,A -155.2474,B 24.9621,C -1.4224,E1 24.8588,E2 241.6978} C_DIS
LIN {X -113.6138,Y -58.5665,Z 142,A -157.141,B 24.963,C -1.4045,E1 24.8564,E2 243.6442} C_DIS
LIN {X -115.7551,Y -54.2117,Z 142,A -158.7158,B 24.9613,C -1.4382,E1 24.8545,E2 245.1472} C_DIS
LIN {X -117.2494,Y -50.8957,Z 142,A -160.3098,B 24.9609,C -1.4447,E1 24.8527,E2 246.7346} C_DIS
LIN {X -118.4653,Y -47.9979,Z 142,A -161.7537,B 24.9608,C -1.4472,E1 24.8512,E2 248.1805} C_DIS
LIN {X -119.5817,Y -45.1456,Z 142,A -163.1892,B 24.9607,C -1.4485,E1 24.8497,E2 249.6211} C_DIS
LIN {X -120.7984,Y -41.7798,Z 142,A -164.6567,B 24.9601,C -1.4596,E1 24.8484,E2 251.0704} C_DIS
LIN {X -121.6159,Y -39.3394,Z 142,A -166.3552,B 24.9613,C -1.4382,E1 24.8469,E2 252.8296} C_DIS
LIN {X -122.7516,Y -35.6361,Z 142,A -167.7212,B 24.96,C -1.4605,E1 24.8458,E2 254.1505} C_DIS
LIN {X -123.8075,Y -31.7748,Z 142,A -169.4923,B 24.9597,C -1.4671,E1 24.8446,E2 255.916} C_DIS
LIN {X -124.6758,Y -28.1755,Z 142,A -170.982,B 24.959,C -1.4801,E1 24.8436,E2 257.3834} C_DIS
Enddeposition()
END
